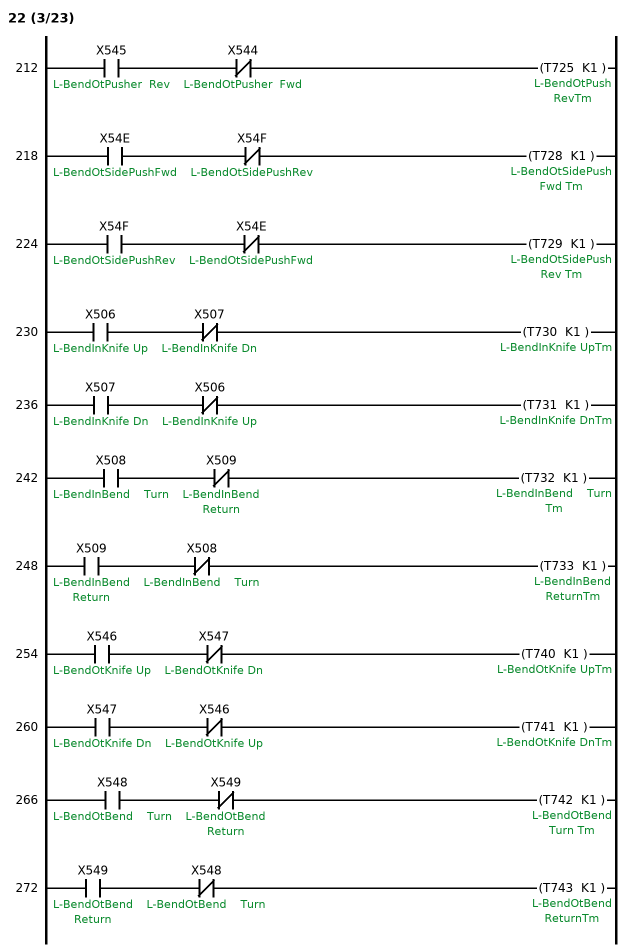
212   LD      X545  ; L-BendOtPusher  Rev
      ANI     X544  ; L-BendOtPusher  Fwd
      OUT     T725 K1  ; L-BendOtPush RevTm
218   LD      X54E  ; L-BendOtSidePushFwd
      ANI     X54F  ; L-BendOtSidePushRev
      OUT     T728 K1  ; L-BendOtSidePushFwd Tm
224   LD      X54F  ; L-BendOtSidePushRev
      ANI     X54E  ; L-BendOtSidePushFwd
      OUT     T729 K1  ; L-BendOtSidePushRev Tm
230   LD      X506  ; L-BendInKnife Up
      ANI     X507  ; L-BendInKnife Dn
      OUT     T730 K1  ; L-BendInKnife UpTm
236   LD      X507  ; L-BendInKnife Dn
      ANI     X506  ; L-BendInKnife Up
      OUT     T731 K1  ; L-BendInKnife DnTm
242   LD      X508  ; L-BendInBend    Turn
      ANI     X509  ; L-BendInBend    Return
      OUT     T732 K1  ; L-BendInBend    Turn Tm
248   LD      X509  ; L-BendInBend    Return
      ANI     X508  ; L-BendInBend    Turn
      OUT     T733 K1  ; L-BendInBend    ReturnTm
254   LD      X546  ; L-BendOtKnife Up
      ANI     X547  ; L-BendOtKnife Dn
      OUT     T740 K1  ; L-BendOtKnife UpTm
260   LD      X547  ; L-BendOtKnife Dn
      ANI     X546  ; L-BendOtKnife Up
      OUT     T741 K1  ; L-BendOtKnife DnTm
266   LD      X548  ; L-BendOtBend    Turn
      ANI     X549  ; L-BendOtBend    Return
      OUT     T742 K1  ; L-BendOtBend    Turn Tm
272   LD      X549  ; L-BendOtBend    Return
      ANI     X548  ; L-BendOtBend    Turn
      OUT     T743 K1  ; L-BendOtBend    ReturnTm
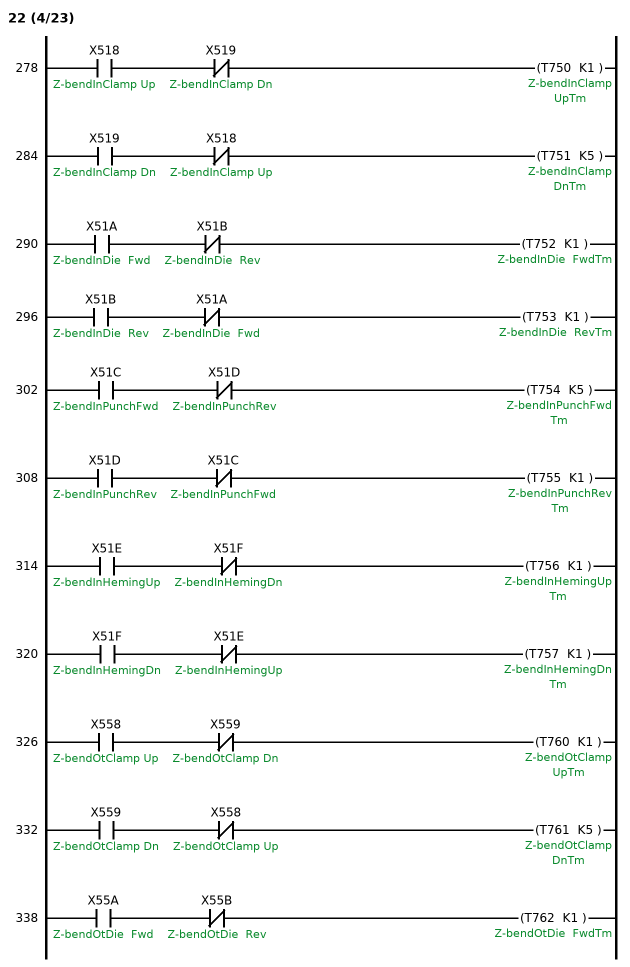
278   LD      X518  ; Z-bendInClamp Up
      ANI     X519  ; Z-bendInClamp Dn
      OUT     T750 K1  ; Z-bendInClamp UpTm
284   LD      X519  ; Z-bendInClamp Dn
      ANI     X518  ; Z-bendInClamp Up
      OUT     T751 K5  ; Z-bendInClamp DnTm
290   LD      X51A  ; Z-bendInDie  Fwd
      ANI     X51B  ; Z-bendInDie  Rev
      OUT     T752 K1  ; Z-bendInDie  FwdTm
296   LD      X51B  ; Z-bendInDie  Rev
      ANI     X51A  ; Z-bendInDie  Fwd
      OUT     T753 K1  ; Z-bendInDie  RevTm
302   LD      X51C  ; Z-bendInPunchFwd
      ANI     X51D  ; Z-bendInPunchRev
      OUT     T754 K5  ; Z-bendInPunchFwdTm
308   LD      X51D  ; Z-bendInPunchRev
      ANI     X51C  ; Z-bendInPunchFwd
      OUT     T755 K1  ; Z-bendInPunchRevTm
314   LD      X51E  ; Z-bendInHemingUp
      ANI     X51F  ; Z-bendInHemingDn
      OUT     T756 K1  ; Z-bendInHemingUpTm
320   LD      X51F  ; Z-bendInHemingDn
      ANI     X51E  ; Z-bendInHemingUp
      OUT     T757 K1  ; Z-bendInHemingDnTm
326   LD      X558  ; Z-bendOtClamp Up
      ANI     X559  ; Z-bendOtClamp Dn
      OUT     T760 K1  ; Z-bendOtClamp UpTm
332   LD      X559  ; Z-bendOtClamp Dn
      ANI     X558  ; Z-bendOtClamp Up
      OUT     T761 K5  ; Z-bendOtClamp DnTm
338   LD      X55A  ; Z-bendOtDie  Fwd
      ANI     X55B  ; Z-bendOtDie  Rev
      OUT     T762 K1  ; Z-bendOtDie  FwdTm
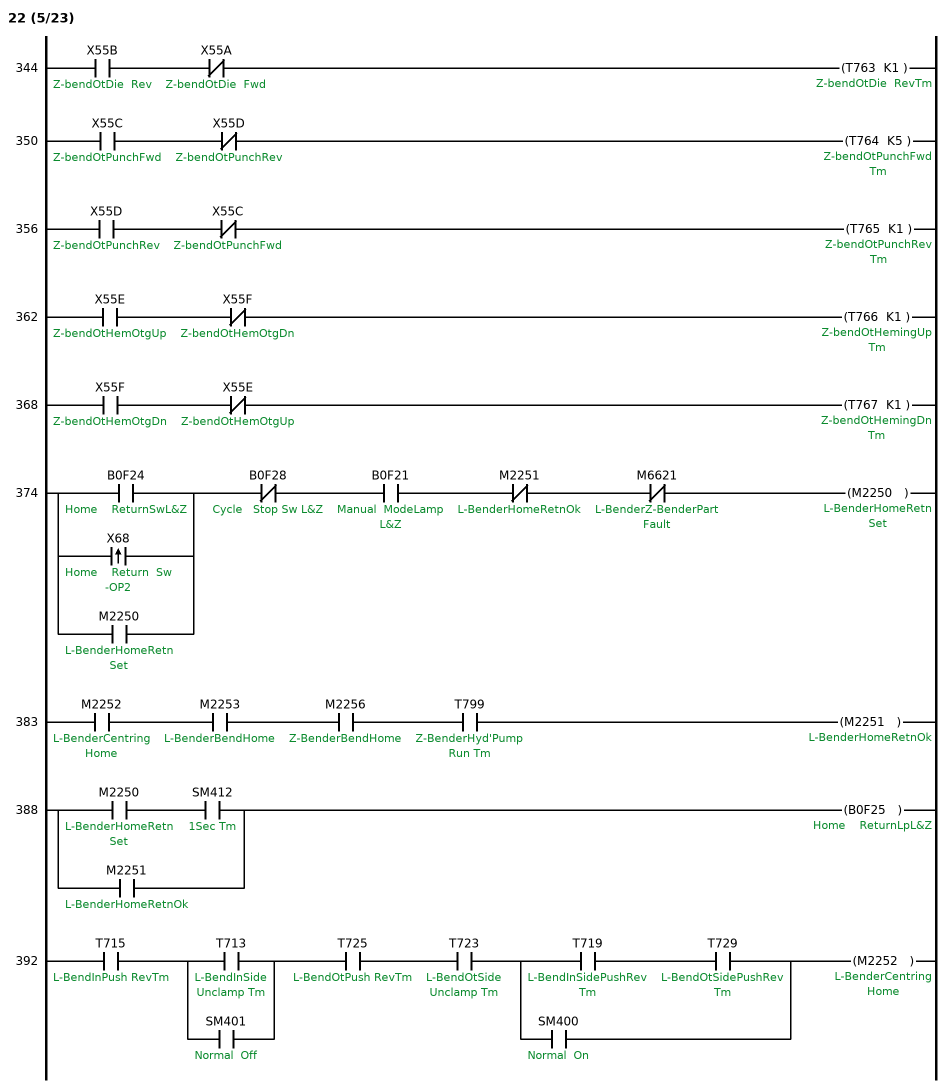
344   LD      X55B  ; Z-bendOtDie  Rev
      ANI     X55A  ; Z-bendOtDie  Fwd
      OUT     T763 K1  ; Z-bendOtDie  RevTm
350   LD      X55C  ; Z-bendOtPunchFwd
      ANI     X55D  ; Z-bendOtPunchRev
      OUT     T764 K5  ; Z-bendOtPunchFwdTm
356   LD      X55D  ; Z-bendOtPunchRev
      ANI     X55C  ; Z-bendOtPunchFwd
      OUT     T765 K1  ; Z-bendOtPunchRevTm
362   LD      X55E  ; Z-bendOtHemOtgUp
      ANI     X55F  ; Z-bendOtHemOtgDn
      OUT     T766 K1  ; Z-bendOtHemingUpTm
368   LD      X55F  ; Z-bendOtHemOtgDn
      ANI     X55E  ; Z-bendOtHemOtgUp
      OUT     T767 K1  ; Z-bendOtHemingDnTm
374   LD      B0F24  ; Home    ReturnSwL&Z
      ORP     X68  ; Home    Return  Sw -OP2
      OR      M2250  ; L-BenderHomeRetnSet
      ANI     B0F28  ; Cycle   Stop Sw L&Z
      AND     B0F21  ; Manual  ModeLampL&Z
      ANI     M2251  ; L-BenderHomeRetnOk
      ANI     M6621  ; L-BenderZ-BenderPart    Fault
      OUT     M2250  ; L-BenderHomeRetnSet
383   LD      M2252  ; L-BenderCentringHome
      AND     M2253  ; L-BenderBendHome
      AND     M2256  ; Z-BenderBendHome
      AND     T799  ; Z-BenderHyd'PumpRun Tm
      OUT     M2251  ; L-BenderHomeRetnOk
388   LD      M2250  ; L-BenderHomeRetnSet
      AND     SM412  ; 1Sec Tm
      OR      M2251  ; L-BenderHomeRetnOk
      OUT     B0F25  ; Home    ReturnLpL&Z
392   LD      T715  ; L-BendInPush RevTm
      LD      T713  ; L-BendInSide    Unclamp Tm
      OR      SM401  ; Normal  Off
      ANB
      AND     T725  ; L-BendOtPush RevTm
      AND     T723  ; L-BendOtSide    Unclamp Tm
      LD      T719  ; L-BendInSidePushRev Tm
      AND     T729  ; L-BendOtSidePushRev Tm
      OR      SM400  ; Normal  On
      ANB
      OUT     M2252  ; L-BenderCentringHome
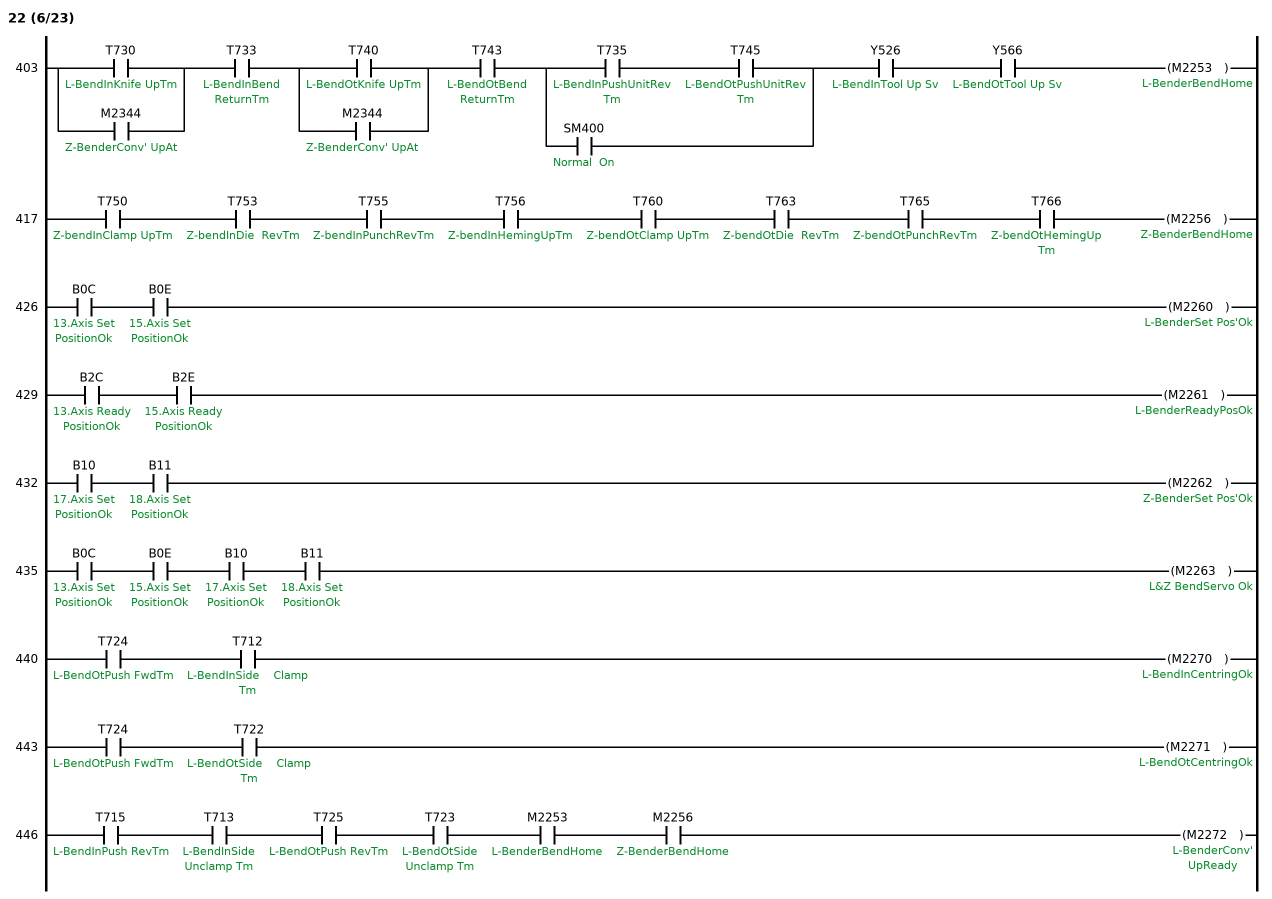
403   LD      T730  ; L-BendInKnife UpTm
      OR      M2344  ; Z-BenderConv' UpAt
      AND     T733  ; L-BendInBend    ReturnTm
      LD      T740  ; L-BendOtKnife UpTm
      OR      M2344  ; Z-BenderConv' UpAt
      ANB
      AND     T743  ; L-BendOtBend    ReturnTm
      LD      T735  ; L-BendInPushUnitRev Tm
      AND     T745  ; L-BendOtPushUnitRev Tm
      OR      SM400  ; Normal  On
      ANB
      AND     Y526  ; L-BendInTool Up Sv
      AND     Y566  ; L-BendOtTool Up Sv
      OUT     M2253  ; L-BenderBendHome
417   LD      T750  ; Z-bendInClamp UpTm
      AND     T753  ; Z-bendInDie  RevTm
      AND     T755  ; Z-bendInPunchRevTm
      AND     T756  ; Z-bendInHemingUpTm
      AND     T760  ; Z-bendOtClamp UpTm
      AND     T763  ; Z-bendOtDie  RevTm
      AND     T765  ; Z-bendOtPunchRevTm
      AND     T766  ; Z-bendOtHemingUpTm
      OUT     M2256  ; Z-BenderBendHome
426   LD      B0C  ; 13.Axis Set     PositionOk
      AND     B0E  ; 15.Axis Set     PositionOk
      OUT     M2260  ; L-BenderSet Pos'Ok
429   LD      B2C  ; 13.Axis Ready   PositionOk
      AND     B2E  ; 15.Axis Ready   PositionOk
      OUT     M2261  ; L-BenderReadyPosOk
432   LD      B10  ; 17.Axis Set     PositionOk
      AND     B11  ; 18.Axis Set     PositionOk
      OUT     M2262  ; Z-BenderSet Pos'Ok
435   LD      B0C  ; 13.Axis Set     PositionOk
      AND     B0E  ; 15.Axis Set     PositionOk
      AND     B10  ; 17.Axis Set     PositionOk
      AND     B11  ; 18.Axis Set     PositionOk
      OUT     M2263  ; L&Z BendServo Ok
440   LD      T724  ; L-BendOtPush FwdTm
      AND     T712  ; L-BendInSide    Clamp Tm
      OUT     M2270  ; L-BendInCentringOk
443   LD      T724  ; L-BendOtPush FwdTm
      AND     T722  ; L-BendOtSide    Clamp Tm
      OUT     M2271  ; L-BendOtCentringOk
446   LD      T715  ; L-BendInPush RevTm
      AND     T713  ; L-BendInSide    Unclamp Tm
      AND     T725  ; L-BendOtPush RevTm
      AND     T723  ; L-BendOtSide    Unclamp Tm
      AND     M2253  ; L-BenderBendHome
      AND     M2256  ; Z-BenderBendHome
      OUT     M2272  ; L-BenderConv' UpReady
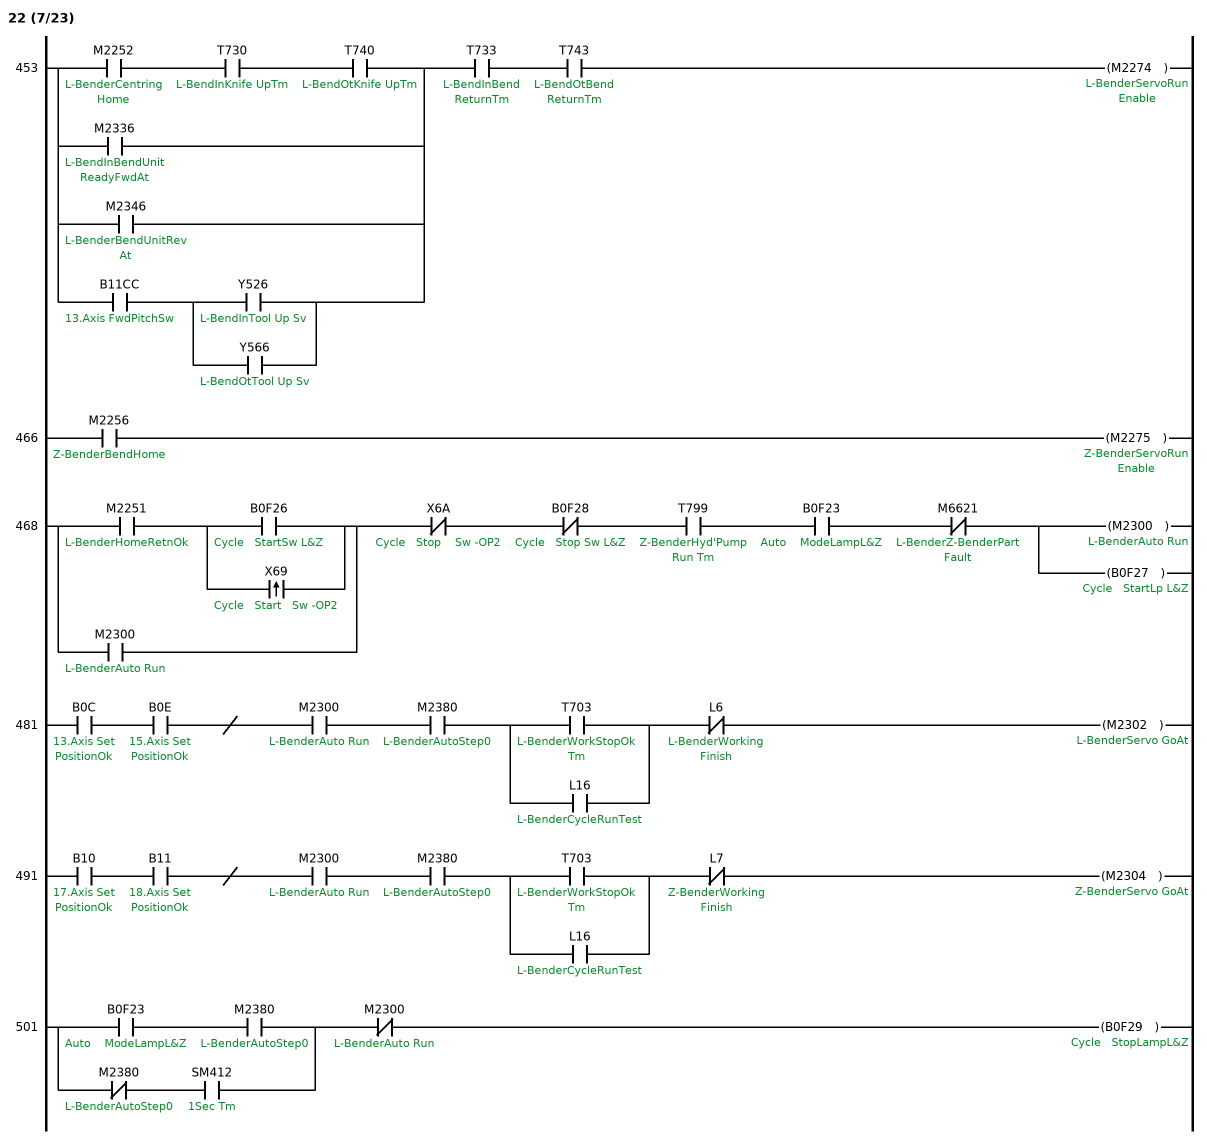
453   LD      M2252  ; L-BenderCentringHome
      AND     T730  ; L-BendInKnife UpTm
      AND     T740  ; L-BendOtKnife UpTm
      OR      M2336  ; L-BendInBendUnitReadyFwdAt
      OR      M2346  ; L-BenderBendUnitRev At
      LD      B11CC  ; 13.Axis FwdPitchSw
      LD      Y526  ; L-BendInTool Up Sv
      OR      Y566  ; L-BendOtTool Up Sv
      ANB
      ORB
      AND     T733  ; L-BendInBend    ReturnTm
      AND     T743  ; L-BendOtBend    ReturnTm
      OUT     M2274  ; L-BenderServoRunEnable
466   LD      M2256  ; Z-BenderBendHome
      OUT     M2275  ; Z-BenderServoRunEnable
468   LD      M2251  ; L-BenderHomeRetnOk
      LD      B0F26  ; Cycle   StartSw L&Z
      ORP     X69  ; Cycle   Start   Sw -OP2
      ANB
      OR      M2300  ; L-BenderAuto Run
      ANI     X6A  ; Cycle   Stop    Sw -OP2
      ANI     B0F28  ; Cycle   Stop Sw L&Z
      AND     T799  ; Z-BenderHyd'PumpRun Tm
      AND     B0F23  ; Auto    ModeLampL&Z
      ANI     M6621  ; L-BenderZ-BenderPart    Fault
      OUT     M2300  ; L-BenderAuto Run
      OUT     B0F27  ; Cycle   StartLp L&Z
481   LD      B0C  ; 13.Axis Set     PositionOk
      AND     B0E  ; 15.Axis Set     PositionOk
      INV
      AND     M2300  ; L-BenderAuto Run
      AND     M2380  ; L-BenderAutoStep0
      LD      T703  ; L-BenderWorkStopOk Tm
      OR      L16  ; L-BenderCycleRunTest
      ANB
      ANI     L6  ; L-BenderWorking Finish
      OUT     M2302  ; L-BenderServo GoAt
491   LD      B10  ; 17.Axis Set     PositionOk
      AND     B11  ; 18.Axis Set     PositionOk
      INV
      AND     M2300  ; L-BenderAuto Run
      AND     M2380  ; L-BenderAutoStep0
      LD      T703  ; L-BenderWorkStopOk Tm
      OR      L16  ; L-BenderCycleRunTest
      ANB
      ANI     L7  ; Z-BenderWorking Finish
      OUT     M2304  ; Z-BenderServo GoAt
501   LD      B0F23  ; Auto    ModeLampL&Z
      AND     M2380  ; L-BenderAutoStep0
      LDI     M2380  ; L-BenderAutoStep0
      AND     SM412  ; 1Sec Tm
      ORB
      ANI     M2300  ; L-BenderAuto Run
      OUT     B0F29  ; Cycle   StopLampL&Z
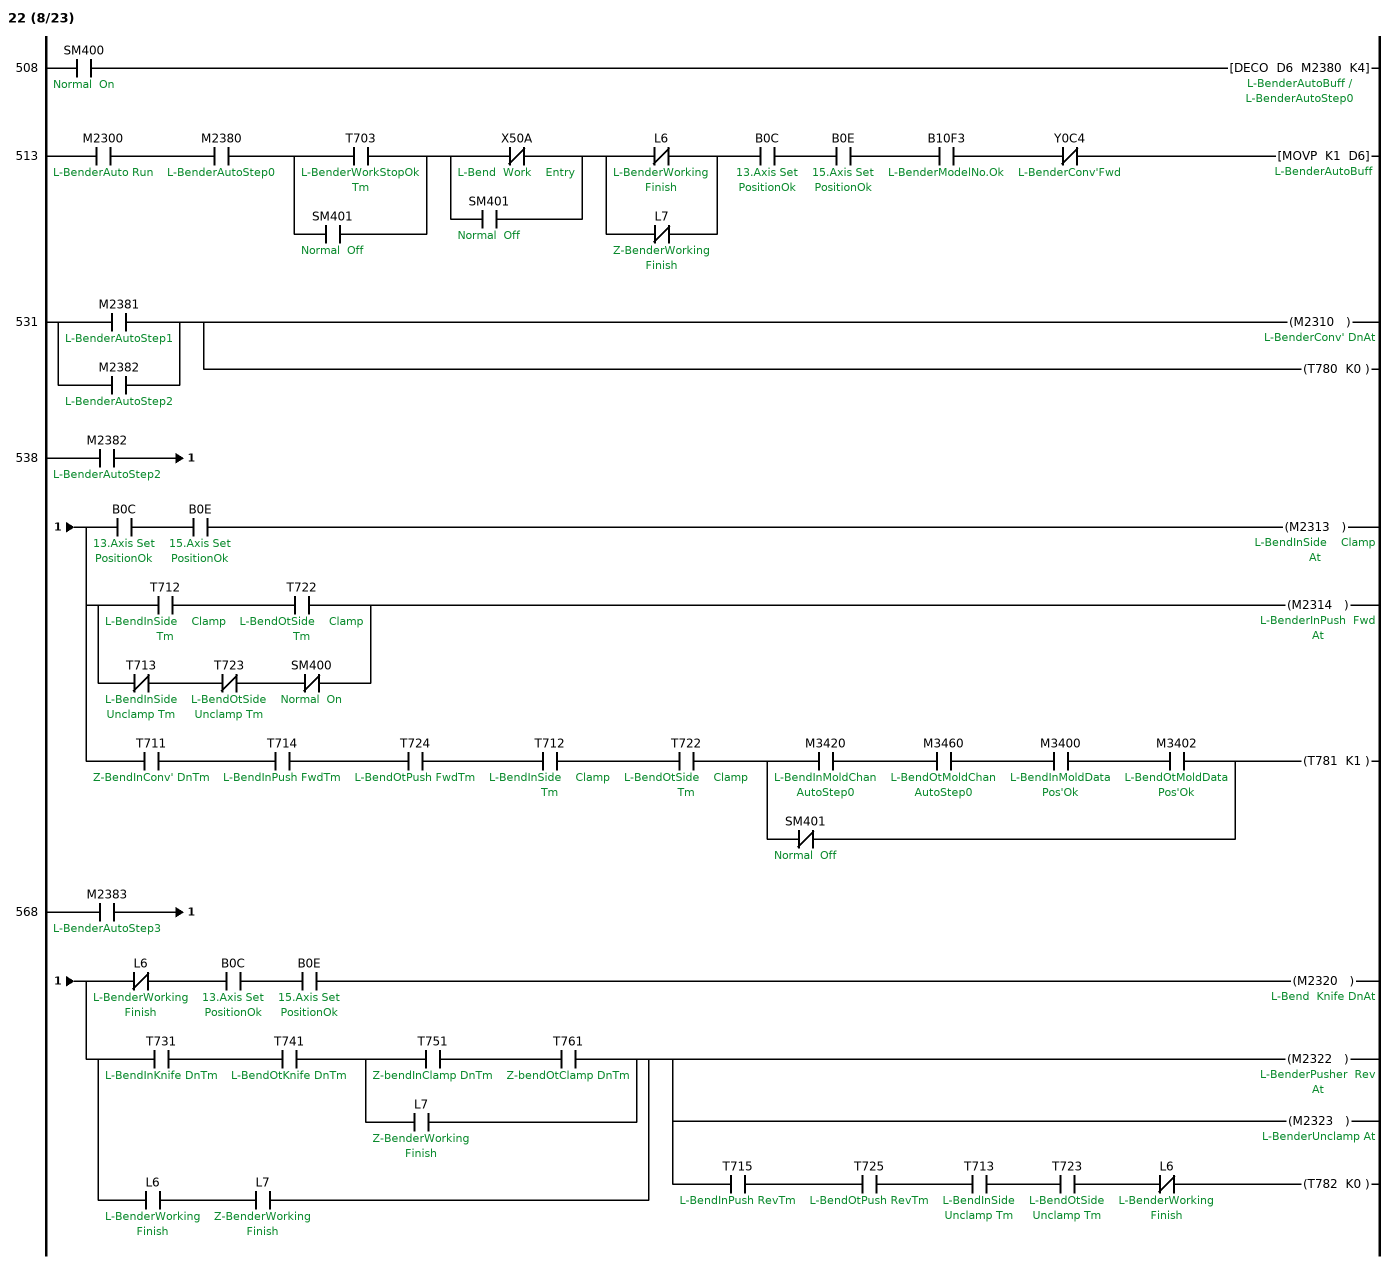
508   LD      SM400  ; Normal  On
      DECO    D6 M2380 K4  ; L-BenderAutoBuff
513   LD      M2300  ; L-BenderAuto Run
      AND     M2380  ; L-BenderAutoStep0
      LD      T703  ; L-BenderWorkStopOk Tm
      OR      SM401  ; Normal  Off
      ANB
      LDI     X50A  ; L-Bend  Work    Entry
      OR      SM401  ; Normal  Off
      ANB
      LDI     L6  ; L-BenderWorking Finish
      ORI     L7  ; Z-BenderWorking Finish
      ANB
      AND     B0C  ; 13.Axis Set     PositionOk
      AND     B0E  ; 15.Axis Set     PositionOk
      AND     B10F3  ; L-BenderModelNo.Ok
      ANI     Y0C4  ; L-BenderConv'Fwd
      MOVP    K1 D6
531   LD      M2381  ; L-BenderAutoStep1
      OR      M2382  ; L-BenderAutoStep2
      OUT     M2310  ; L-BenderConv' DnAt
      OUT     T780 K0
538   LD      M2382  ; L-BenderAutoStep2
      MPS
      AND     B0C  ; 13.Axis Set     PositionOk
      AND     B0E  ; 15.Axis Set     PositionOk
      OUT     M2313  ; L-BendInSide    Clamp At
      MRD
      LD      T712  ; L-BendInSide    Clamp Tm
      AND     T722  ; L-BendOtSide    Clamp Tm
      LDI     T713  ; L-BendInSide    Unclamp Tm
      ANI     T723  ; L-BendOtSide    Unclamp Tm
      ANI     SM400  ; Normal  On
      ORB
      ANB
      OUT     M2314  ; L-BenderInPush  Fwd At
      MPP
      AND     T711  ; Z-BendInConv' DnTm
      AND     T714  ; L-BendInPush FwdTm
      AND     T724  ; L-BendOtPush FwdTm
      AND     T712  ; L-BendInSide    Clamp Tm
      AND     T722  ; L-BendOtSide    Clamp Tm
      LD      M3420  ; L-BendInMoldChanAutoStep0
      AND     M3460  ; L-BendOtMoldChanAutoStep0
      AND     M3400  ; L-BendInMoldDataPos'Ok
      AND     M3402  ; L-BendOtMoldDataPos'Ok
      ORI     SM401  ; Normal  Off
      ANB
      OUT     T781 K1
568   LD      M2383  ; L-BenderAutoStep3
      MPS
      ANI     L6  ; L-BenderWorking Finish
      AND     B0C  ; 13.Axis Set     PositionOk
      AND     B0E  ; 15.Axis Set     PositionOk
      OUT     M2320  ; L-Bend  Knife DnAt
      MPP
      LD      T731  ; L-BendInKnife DnTm
      AND     T741  ; L-BendOtKnife DnTm
      LD      T751  ; Z-bendInClamp DnTm
      AND     T761  ; Z-bendOtClamp DnTm
      OR      L7  ; Z-BenderWorking Finish
      ANB
      LD      L6  ; L-BenderWorking Finish
      AND     L7  ; Z-BenderWorking Finish
      ORB
      ANB
      OUT     M2322  ; L-BenderPusher  Rev At
      OUT     M2323  ; L-BenderUnclamp At
      AND     T715  ; L-BendInPush RevTm
      AND     T725  ; L-BendOtPush RevTm
      AND     T713  ; L-BendInSide    Unclamp Tm
      AND     T723  ; L-BendOtSide    Unclamp Tm
      ANI     L6  ; L-BenderWorking Finish
      OUT     T782 K0
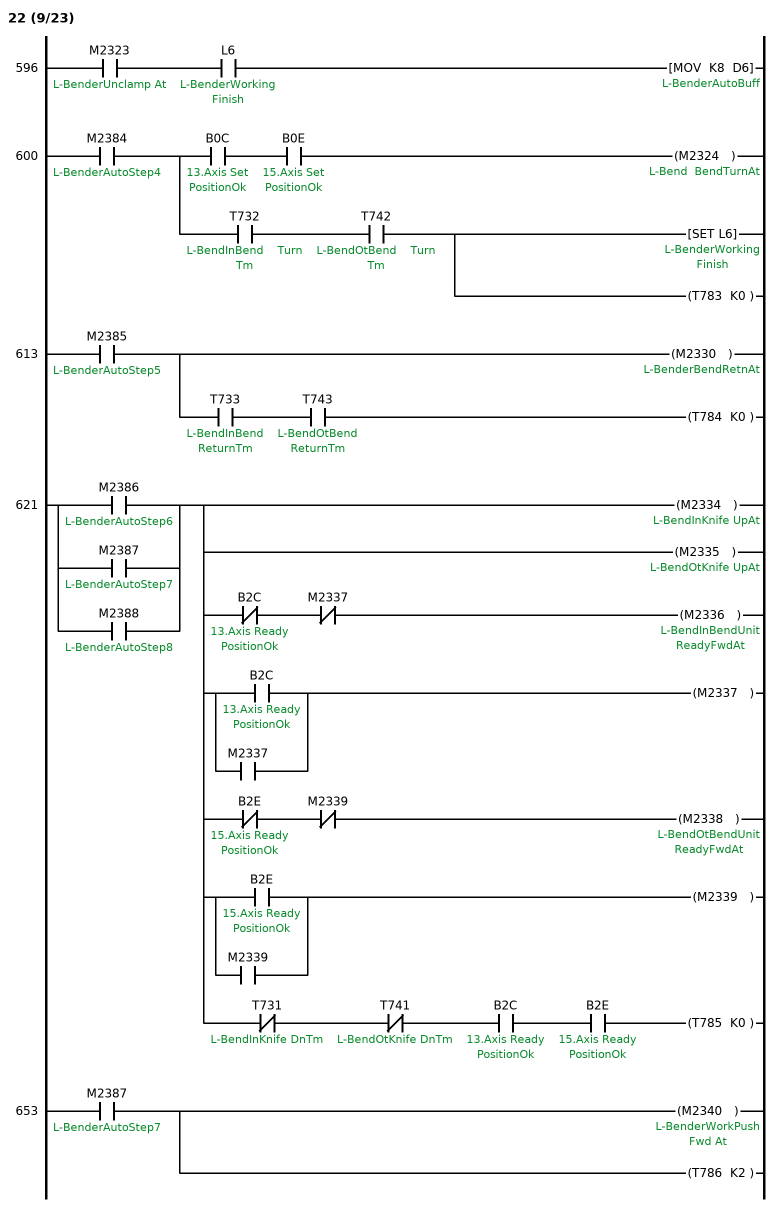
596   LD      M2323  ; L-BenderUnclamp At
      AND     L6  ; L-BenderWorking Finish
      MOV     K8 D6
600   LD      M2384  ; L-BenderAutoStep4
      MPS
      AND     B0C  ; 13.Axis Set     PositionOk
      AND     B0E  ; 15.Axis Set     PositionOk
      OUT     M2324  ; L-Bend  BendTurnAt
      MPP
      AND     T732  ; L-BendInBend    Turn Tm
      AND     T742  ; L-BendOtBend    Turn Tm
      SET     L6  ; L-BenderWorking Finish
      OUT     T783 K0
613   LD      M2385  ; L-BenderAutoStep5
      OUT     M2330  ; L-BenderBendRetnAt
      AND     T733  ; L-BendInBend    ReturnTm
      AND     T743  ; L-BendOtBend    ReturnTm
      OUT     T784 K0
621   LD      M2386  ; L-BenderAutoStep6
      OR      M2387  ; L-BenderAutoStep7
      OR      M2388  ; L-BenderAutoStep8
      OUT     M2334  ; L-BendInKnife UpAt
      OUT     M2335  ; L-BendOtKnife UpAt
      MPS
      ANI     B2C  ; 13.Axis Ready   PositionOk
      ANI     M2337
      OUT     M2336  ; L-BendInBendUnitReadyFwdAt
      MRD
      LD      B2C  ; 13.Axis Ready   PositionOk
      OR      M2337
      ANB
      OUT     M2337
      MRD
      ANI     B2E  ; 15.Axis Ready   PositionOk
      ANI     M2339
      OUT     M2338  ; L-BendOtBendUnitReadyFwdAt
      MRD
      LD      B2E  ; 15.Axis Ready   PositionOk
      OR      M2339
      ANB
      OUT     M2339
      MPP
      ANI     T731  ; L-BendInKnife DnTm
      ANI     T741  ; L-BendOtKnife DnTm
      AND     B2C  ; 13.Axis Ready   PositionOk
      AND     B2E  ; 15.Axis Ready   PositionOk
      OUT     T785 K0
653   LD      M2387  ; L-BenderAutoStep7
      OUT     M2340  ; L-BenderWorkPushFwd At
      OUT     T786 K2
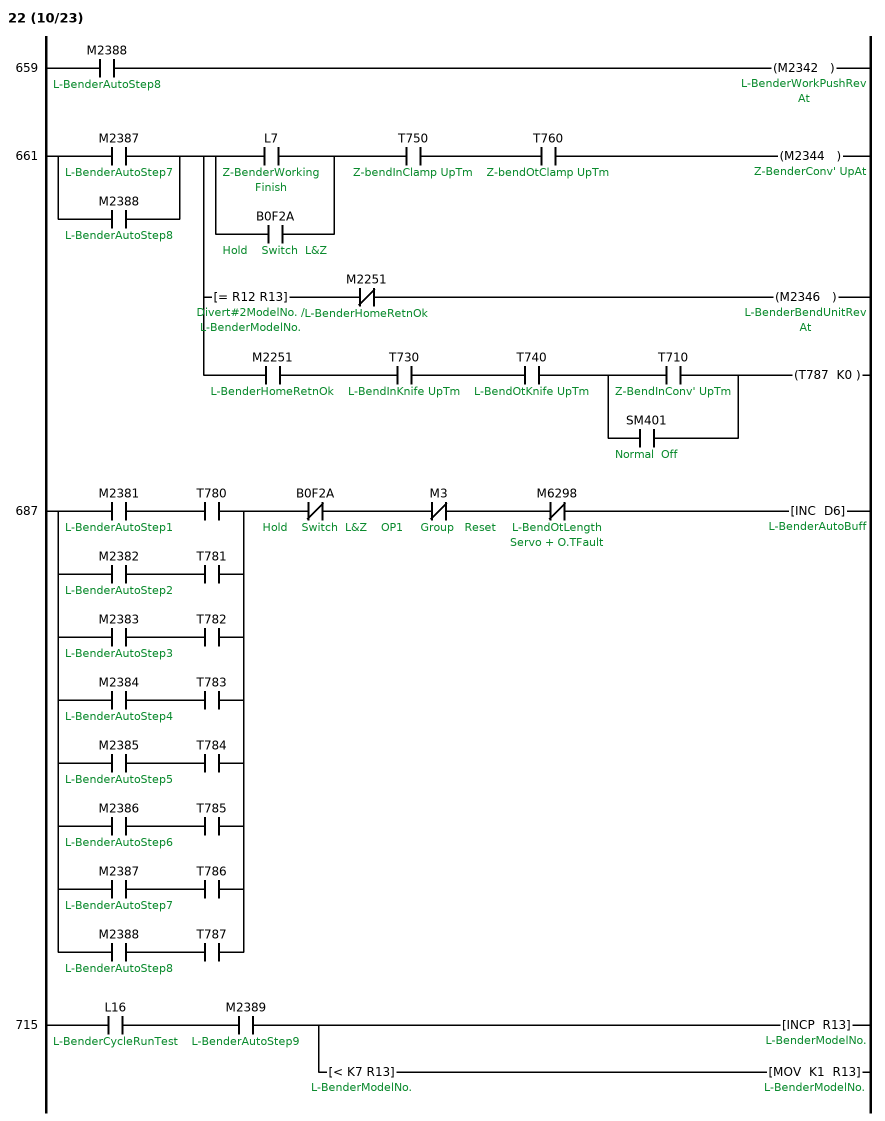
659   LD      M2388  ; L-BenderAutoStep8
      OUT     M2342  ; L-BenderWorkPushRev At
661   LD      M2387  ; L-BenderAutoStep7
      OR      M2388  ; L-BenderAutoStep8
      MPS
      LD      L7  ; Z-BenderWorking Finish
      OR      B0F2A  ; Hold    Switch  L&Z
      ANB
      AND     T750  ; Z-bendInClamp UpTm
      AND     T760  ; Z-bendOtClamp UpTm
      OUT     M2344  ; Z-BenderConv' UpAt
      MRD
      AND=    R12 R13  ; Divert#2ModelNo. / L-BenderModelNo.
      ANI     M2251  ; L-BenderHomeRetnOk
      OUT     M2346  ; L-BenderBendUnitRev At
      MPP
      AND     M2251  ; L-BenderHomeRetnOk
      AND     T730  ; L-BendInKnife UpTm
      AND     T740  ; L-BendOtKnife UpTm
      LD      T710  ; Z-BendInConv' UpTm
      OR      SM401  ; Normal  Off
      ANB
      OUT     T787 K0
687   LD      M2381  ; L-BenderAutoStep1
      AND     T780
      LD      M2382  ; L-BenderAutoStep2
      AND     T781
      ORB
      LD      M2383  ; L-BenderAutoStep3
      AND     T782
      ORB
      LD      M2384  ; L-BenderAutoStep4
      AND     T783
      ORB
      LD      M2385  ; L-BenderAutoStep5
      AND     T784
      ORB
      LD      M2386  ; L-BenderAutoStep6
      AND     T785
      ORB
      LD      M2387  ; L-BenderAutoStep7
      AND     T786
      ORB
      LD      M2388  ; L-BenderAutoStep8
      AND     T787
      ORB
      ANI     B0F2A  ; Hold    Switch  L&Z
      ANI     M3  ; OP1     Group   Reset
      ANI     M6298  ; L-BendOtLength  Servo + O.TFault
      INC     D6
715   LD      L16  ; L-BenderCycleRunTest
      AND     M2389  ; L-BenderAutoStep9
      INCP    R13
      AND<    K7 R13  ; L-BenderModelNo.
      MOV     K1 R13
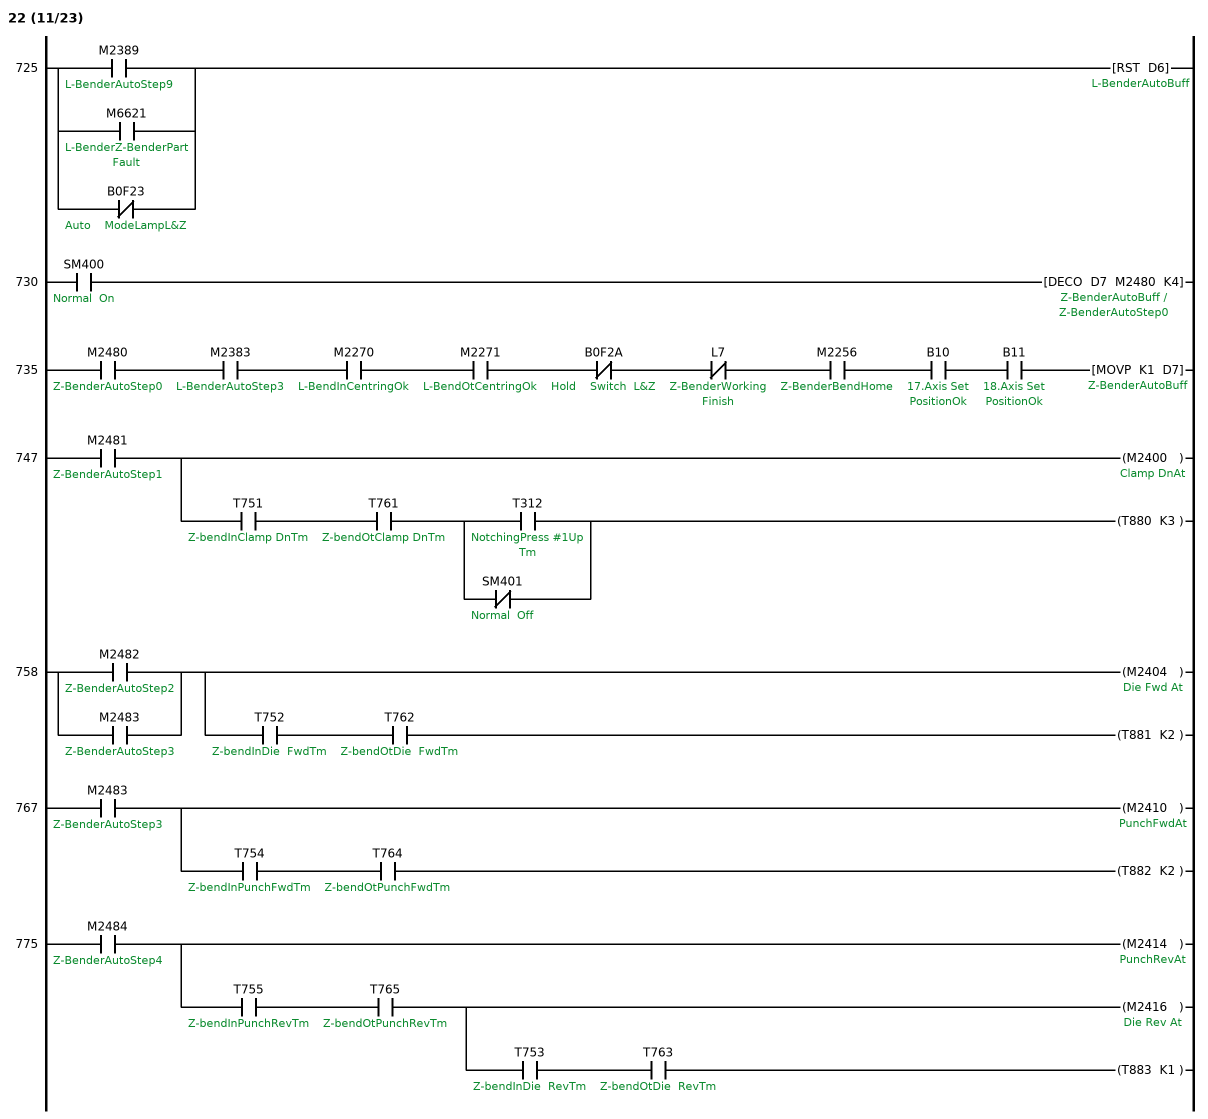
725   LD      M2389  ; L-BenderAutoStep9
      OR      M6621  ; L-BenderZ-BenderPart    Fault
      ORI     B0F23  ; Auto    ModeLampL&Z
      RST     D6  ; L-BenderAutoBuff
730   LD      SM400  ; Normal  On
      DECO    D7 M2480 K4  ; Z-BenderAutoBuff / Z-BenderAutoStep0
735   LD      M2480  ; Z-BenderAutoStep0
      AND     M2383  ; L-BenderAutoStep3
      AND     M2270  ; L-BendInCentringOk
      AND     M2271  ; L-BendOtCentringOk
      ANI     B0F2A  ; Hold    Switch  L&Z
      ANI     L7  ; Z-BenderWorking Finish
      AND     M2256  ; Z-BenderBendHome
      AND     B10  ; 17.Axis Set     PositionOk
      AND     B11  ; 18.Axis Set     PositionOk
      MOVP    K1 D7
747   LD      M2481  ; Z-BenderAutoStep1
      OUT     M2400  ; Clamp DnAt
      AND     T751  ; Z-bendInClamp DnTm
      AND     T761  ; Z-bendOtClamp DnTm
      LD      T312  ; NotchingPress #1Up Tm
      ORI     SM401  ; Normal  Off
      ANB
      OUT     T880 K3
758   LD      M2482  ; Z-BenderAutoStep2
      OR      M2483  ; Z-BenderAutoStep3
      OUT     M2404  ; Die Fwd At
      AND     T752  ; Z-bendInDie  FwdTm
      AND     T762  ; Z-bendOtDie  FwdTm
      OUT     T881 K2
767   LD      M2483  ; Z-BenderAutoStep3
      OUT     M2410  ; PunchFwdAt
      AND     T754  ; Z-bendInPunchFwdTm
      AND     T764  ; Z-bendOtPunchFwdTm
      OUT     T882 K2
775   LD      M2484  ; Z-BenderAutoStep4
      OUT     M2414  ; PunchRevAt
      AND     T755  ; Z-bendInPunchRevTm
      AND     T765  ; Z-bendOtPunchRevTm
      OUT     M2416  ; Die Rev At
      AND     T753  ; Z-bendInDie  RevTm
      AND     T763  ; Z-bendOtDie  RevTm
      OUT     T883 K1
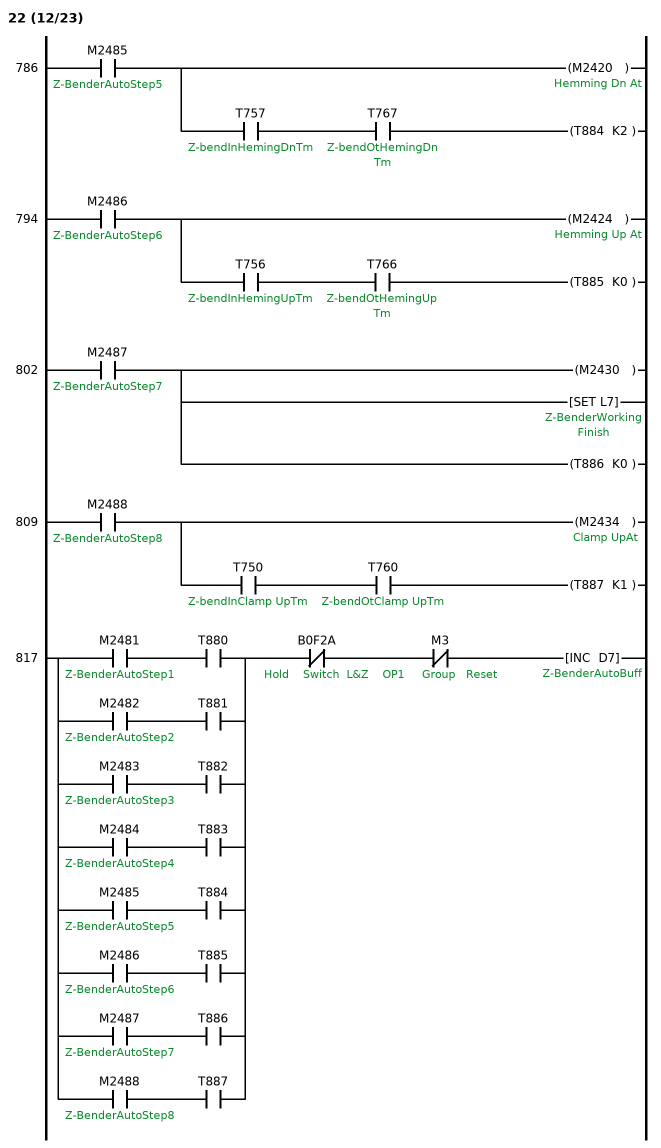
786   LD      M2485  ; Z-BenderAutoStep5
      OUT     M2420  ; Hemming Dn At
      AND     T757  ; Z-bendInHemingDnTm
      AND     T767  ; Z-bendOtHemingDnTm
      OUT     T884 K2
794   LD      M2486  ; Z-BenderAutoStep6
      OUT     M2424  ; Hemming Up At
      AND     T756  ; Z-bendInHemingUpTm
      AND     T766  ; Z-bendOtHemingUpTm
      OUT     T885 K0
802   LD      M2487  ; Z-BenderAutoStep7
      OUT     M2430
      SET     L7  ; Z-BenderWorking Finish
      OUT     T886 K0
809   LD      M2488  ; Z-BenderAutoStep8
      OUT     M2434  ; Clamp UpAt
      AND     T750  ; Z-bendInClamp UpTm
      AND     T760  ; Z-bendOtClamp UpTm
      OUT     T887 K1
817   LD      M2481  ; Z-BenderAutoStep1
      AND     T880
      LD      M2482  ; Z-BenderAutoStep2
      AND     T881
      ORB
      LD      M2483  ; Z-BenderAutoStep3
      AND     T882
      ORB
      LD      M2484  ; Z-BenderAutoStep4
      AND     T883
      ORB
      LD      M2485  ; Z-BenderAutoStep5
      AND     T884
      ORB
      LD      M2486  ; Z-BenderAutoStep6
      AND     T885
      ORB
      LD      M2487  ; Z-BenderAutoStep7
      AND     T886
      ORB
      LD      M2488  ; Z-BenderAutoStep8
      AND     T887
      ORB
      ANI     B0F2A  ; Hold    Switch  L&Z
      ANI     M3  ; OP1     Group   Reset
      INC     D7
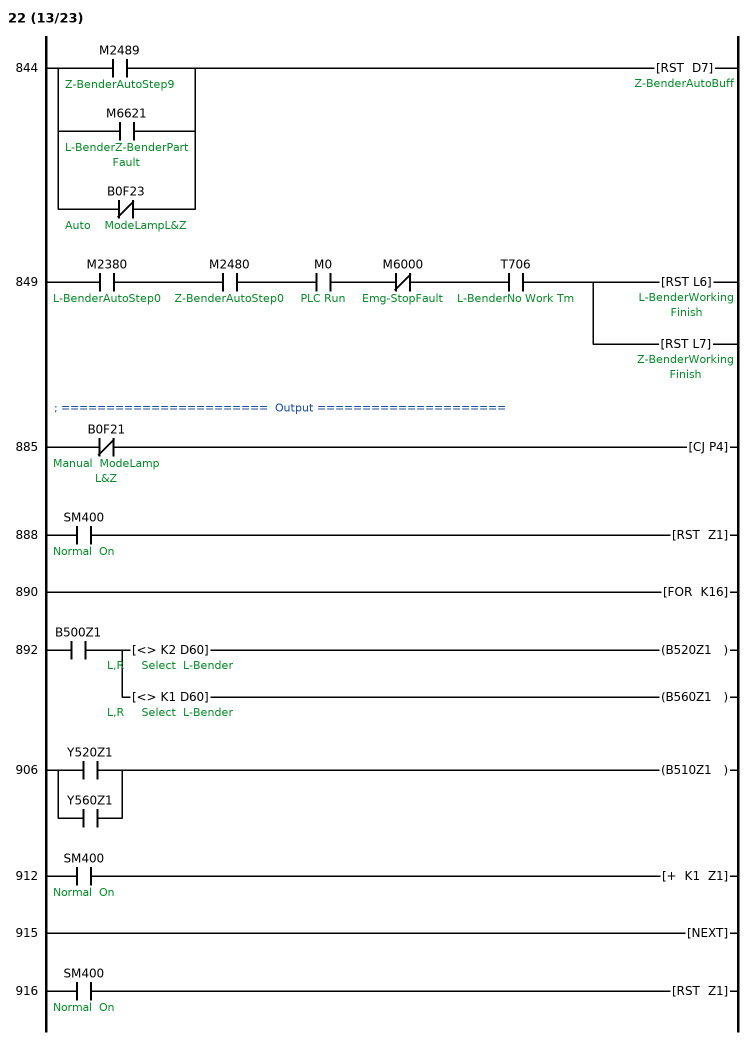
844   LD      M2489  ; Z-BenderAutoStep9
      OR      M6621  ; L-BenderZ-BenderPart    Fault
      ORI     B0F23  ; Auto    ModeLampL&Z
      RST     D7  ; Z-BenderAutoBuff
849   LD      M2380  ; L-BenderAutoStep0
      AND     M2480  ; Z-BenderAutoStep0
      AND     M0  ; PLC Run
      ANI     M6000  ; Emg-StopFault
      AND     T706  ; L-BenderNo Work Tm
      RST     L6  ; L-BenderWorking Finish
      RST     L7  ; Z-BenderWorking Finish
; =======================  Output =====================
885   LDI     B0F21  ; Manual  ModeLampL&Z
      CJ      P4
888   LD      SM400  ; Normal  On
      RST     Z1
890   FOR     K16
892   LD      B500Z1
      MPS
      AND<>   K2 D60  ; L,R     Select  L-Bender
      OUT     B520Z1
      MPP
      AND<>   K1 D60  ; L,R     Select  L-Bender
      OUT     B560Z1
906   LD      Y520Z1
      OR      Y560Z1
      OUT     B510Z1
912   LD      SM400  ; Normal  On
      +       K1 Z1
915   NEXT
916   LD      SM400  ; Normal  On
      RST     Z1
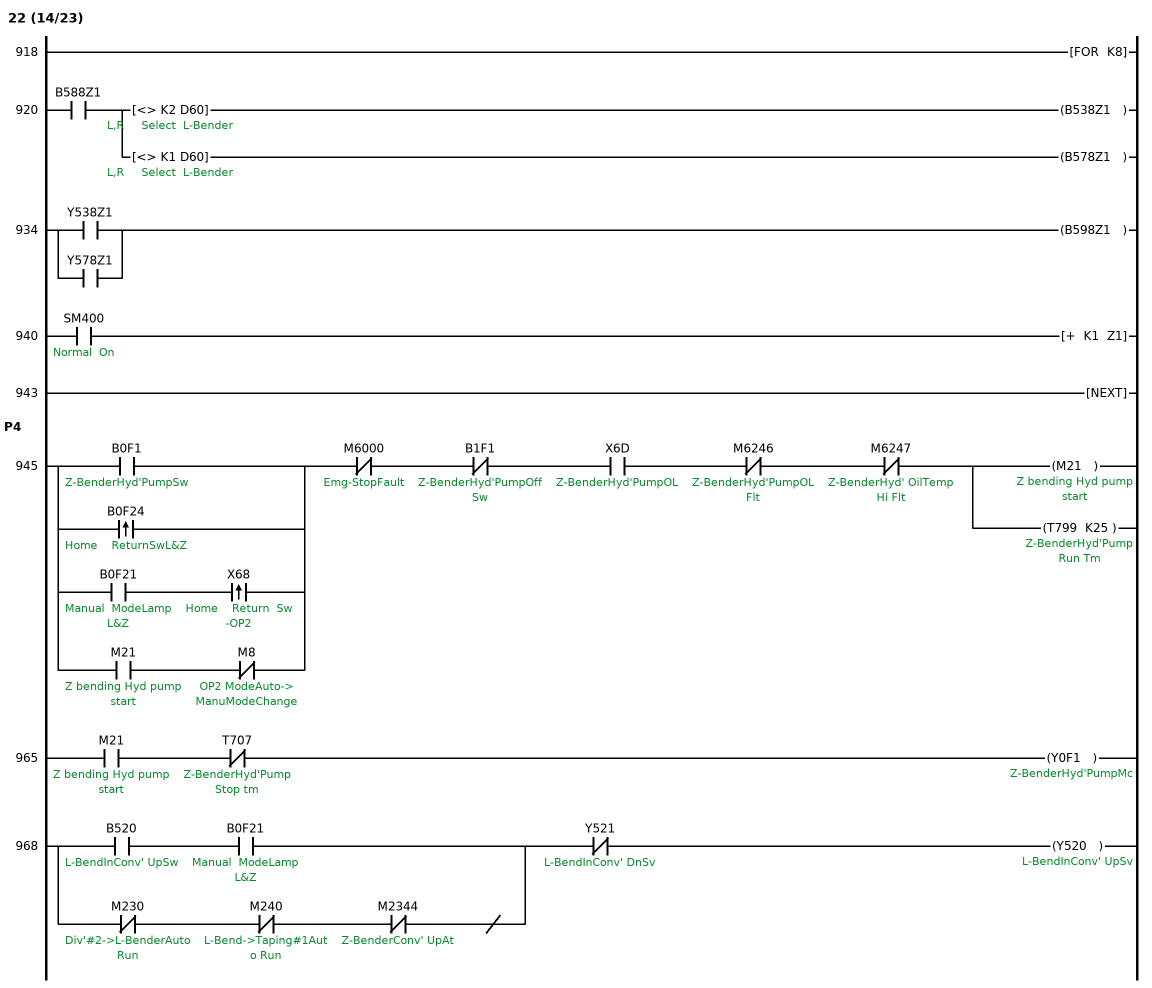
918   FOR     K8
920   LD      B588Z1
      MPS
      AND<>   K2 D60  ; L,R     Select  L-Bender
      OUT     B538Z1
      MPP
      AND<>   K1 D60  ; L,R     Select  L-Bender
      OUT     B578Z1
934   LD      Y538Z1
      OR      Y578Z1
      OUT     B598Z1
940   LD      SM400  ; Normal  On
      +       K1 Z1
943   NEXT
      P4
945   LD      B0F1  ; Z-BenderHyd'PumpSw
      ORP     B0F24  ; Home    ReturnSwL&Z
      LD      B0F21  ; Manual  ModeLampL&Z
      ANDP    X68  ; Home    Return  Sw -OP2
      ORB
      LD      M21  ; Z bending Hyd pump start
      ANI     M8  ; OP2 ModeAuto->  ManuModeChange
      ORB
      ANI     M6000  ; Emg-StopFault
      ANI     B1F1  ; Z-BenderHyd'PumpOff Sw
      AND     X6D  ; Z-BenderHyd'PumpOL
      ANI     M6246  ; Z-BenderHyd'PumpOL Flt
      ANI     M6247  ; Z-BenderHyd' OilTemp Hi Flt
      OUT     M21  ; Z bending Hyd pump start
      OUT     T799 K25  ; Z-BenderHyd'PumpRun Tm
965   LD      M21  ; Z bending Hyd pump start
      ANI     T707  ; Z-BenderHyd'PumpStop tm
      OUT     Y0F1  ; Z-BenderHyd'PumpMc
968   LD      B520  ; L-BendInConv' UpSw
      AND     B0F21  ; Manual  ModeLampL&Z
      LDI     M230  ; Div'#2->L-BenderAuto Run
      ANI     M240  ; L-Bend->Taping#1Auto Run
      ANI     M2344  ; Z-BenderConv' UpAt
      INV
      ORB
      ANI     Y521  ; L-BendInConv' DnSv
      OUT     Y520  ; L-BendInConv' UpSv
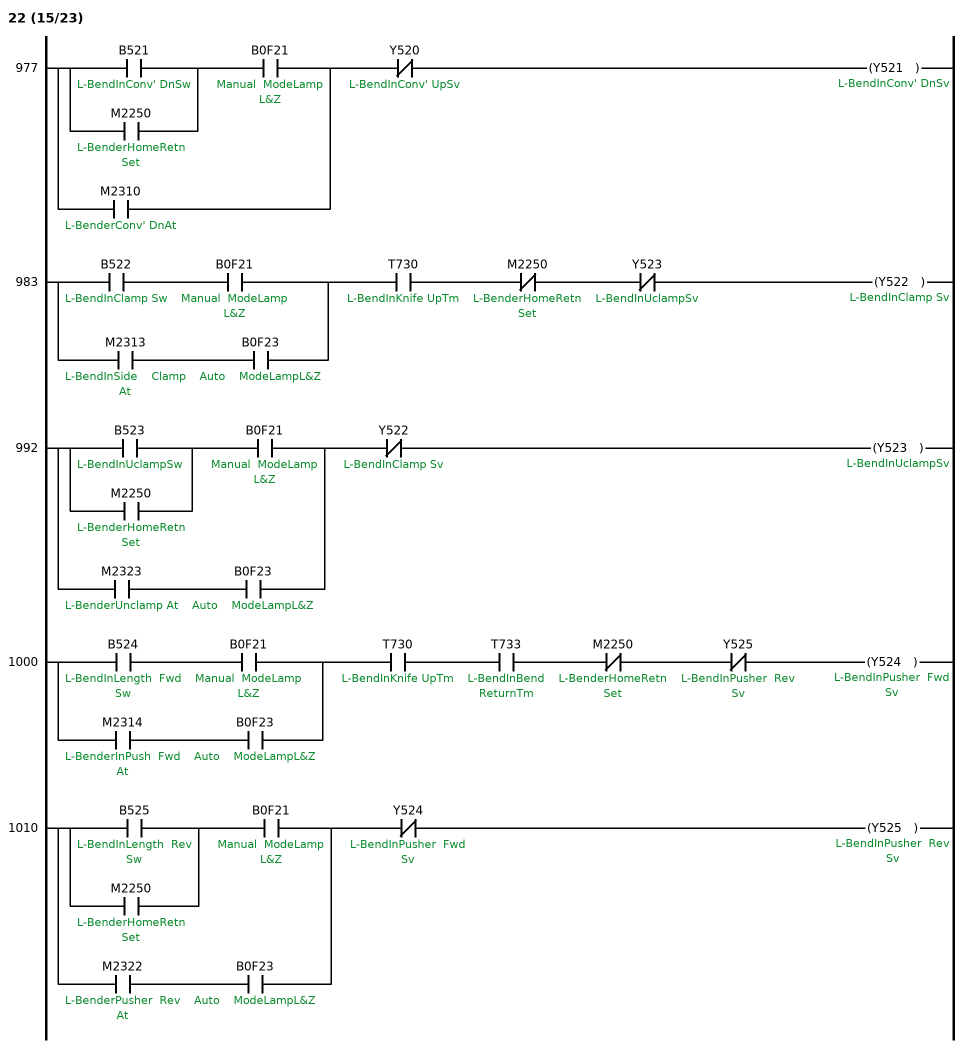
977   LD      B521  ; L-BendInConv' DnSw
      OR      M2250  ; L-BenderHomeRetnSet
      AND     B0F21  ; Manual  ModeLampL&Z
      OR      M2310  ; L-BenderConv' DnAt
      ANI     Y520  ; L-BendInConv' UpSv
      OUT     Y521  ; L-BendInConv' DnSv
983   LD      B522  ; L-BendInClamp Sw
      AND     B0F21  ; Manual  ModeLampL&Z
      LD      M2313  ; L-BendInSide    Clamp At
      AND     B0F23  ; Auto    ModeLampL&Z
      ORB
      AND     T730  ; L-BendInKnife UpTm
      ANI     M2250  ; L-BenderHomeRetnSet
      ANI     Y523  ; L-BendInUclampSv
      OUT     Y522  ; L-BendInClamp Sv
992   LD      B523  ; L-BendInUclampSw
      OR      M2250  ; L-BenderHomeRetnSet
      AND     B0F21  ; Manual  ModeLampL&Z
      LD      M2323  ; L-BenderUnclamp At
      AND     B0F23  ; Auto    ModeLampL&Z
      ORB
      ANI     Y522  ; L-BendInClamp Sv
      OUT     Y523  ; L-BendInUclampSv
1000  LD      B524  ; L-BendInLength  Fwd Sw
      AND     B0F21  ; Manual  ModeLampL&Z
      LD      M2314  ; L-BenderInPush  Fwd At
      AND     B0F23  ; Auto    ModeLampL&Z
      ORB
      AND     T730  ; L-BendInKnife UpTm
      AND     T733  ; L-BendInBend    ReturnTm
      ANI     M2250  ; L-BenderHomeRetnSet
      ANI     Y525  ; L-BendInPusher  Rev Sv
      OUT     Y524  ; L-BendInPusher  Fwd Sv
1010  LD      B525  ; L-BendInLength  Rev Sw
      OR      M2250  ; L-BenderHomeRetnSet
      AND     B0F21  ; Manual  ModeLampL&Z
      LD      M2322  ; L-BenderPusher  Rev At
      AND     B0F23  ; Auto    ModeLampL&Z
      ORB
      ANI     Y524  ; L-BendInPusher  Fwd Sv
      OUT     Y525  ; L-BendInPusher  Rev Sv
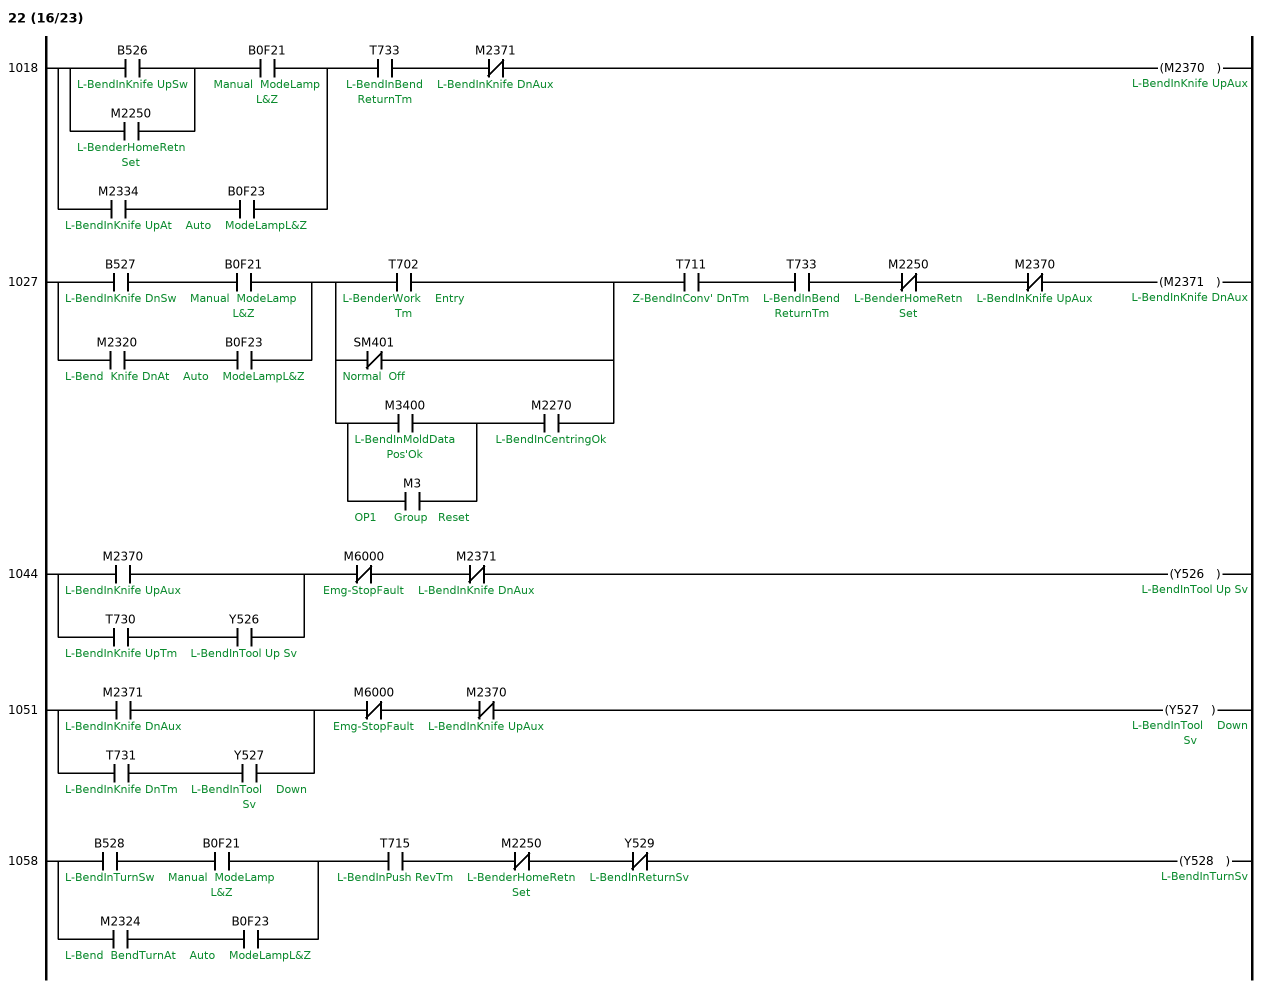
1018  LD      B526  ; L-BendInKnife UpSw
      OR      M2250  ; L-BenderHomeRetnSet
      AND     B0F21  ; Manual  ModeLampL&Z
      LD      M2334  ; L-BendInKnife UpAt
      AND     B0F23  ; Auto    ModeLampL&Z
      ORB
      AND     T733  ; L-BendInBend    ReturnTm
      ANI     M2371  ; L-BendInKnife DnAux
      OUT     M2370  ; L-BendInKnife UpAux
1027  LD      B527  ; L-BendInKnife DnSw
      AND     B0F21  ; Manual  ModeLampL&Z
      LD      M2320  ; L-Bend  Knife DnAt
      AND     B0F23  ; Auto    ModeLampL&Z
      ORB
      LD      T702  ; L-BenderWork    Entry Tm
      ORI     SM401  ; Normal  Off
      LD      M3400  ; L-BendInMoldDataPos'Ok
      OR      M3  ; OP1     Group   Reset
      AND     M2270  ; L-BendInCentringOk
      ORB
      ANB
      AND     T711  ; Z-BendInConv' DnTm
      AND     T733  ; L-BendInBend    ReturnTm
      ANI     M2250  ; L-BenderHomeRetnSet
      ANI     M2370  ; L-BendInKnife UpAux
      OUT     M2371  ; L-BendInKnife DnAux
1044  LD      M2370  ; L-BendInKnife UpAux
      LD      T730  ; L-BendInKnife UpTm
      AND     Y526  ; L-BendInTool Up Sv
      ORB
      ANI     M6000  ; Emg-StopFault
      ANI     M2371  ; L-BendInKnife DnAux
      OUT     Y526  ; L-BendInTool Up Sv
1051  LD      M2371  ; L-BendInKnife DnAux
      LD      T731  ; L-BendInKnife DnTm
      AND     Y527  ; L-BendInTool    Down Sv
      ORB
      ANI     M6000  ; Emg-StopFault
      ANI     M2370  ; L-BendInKnife UpAux
      OUT     Y527  ; L-BendInTool    Down Sv
1058  LD      B528  ; L-BendInTurnSw
      AND     B0F21  ; Manual  ModeLampL&Z
      LD      M2324  ; L-Bend  BendTurnAt
      AND     B0F23  ; Auto    ModeLampL&Z
      ORB
      AND     T715  ; L-BendInPush RevTm
      ANI     M2250  ; L-BenderHomeRetnSet
      ANI     Y529  ; L-BendInReturnSv
      OUT     Y528  ; L-BendInTurnSv
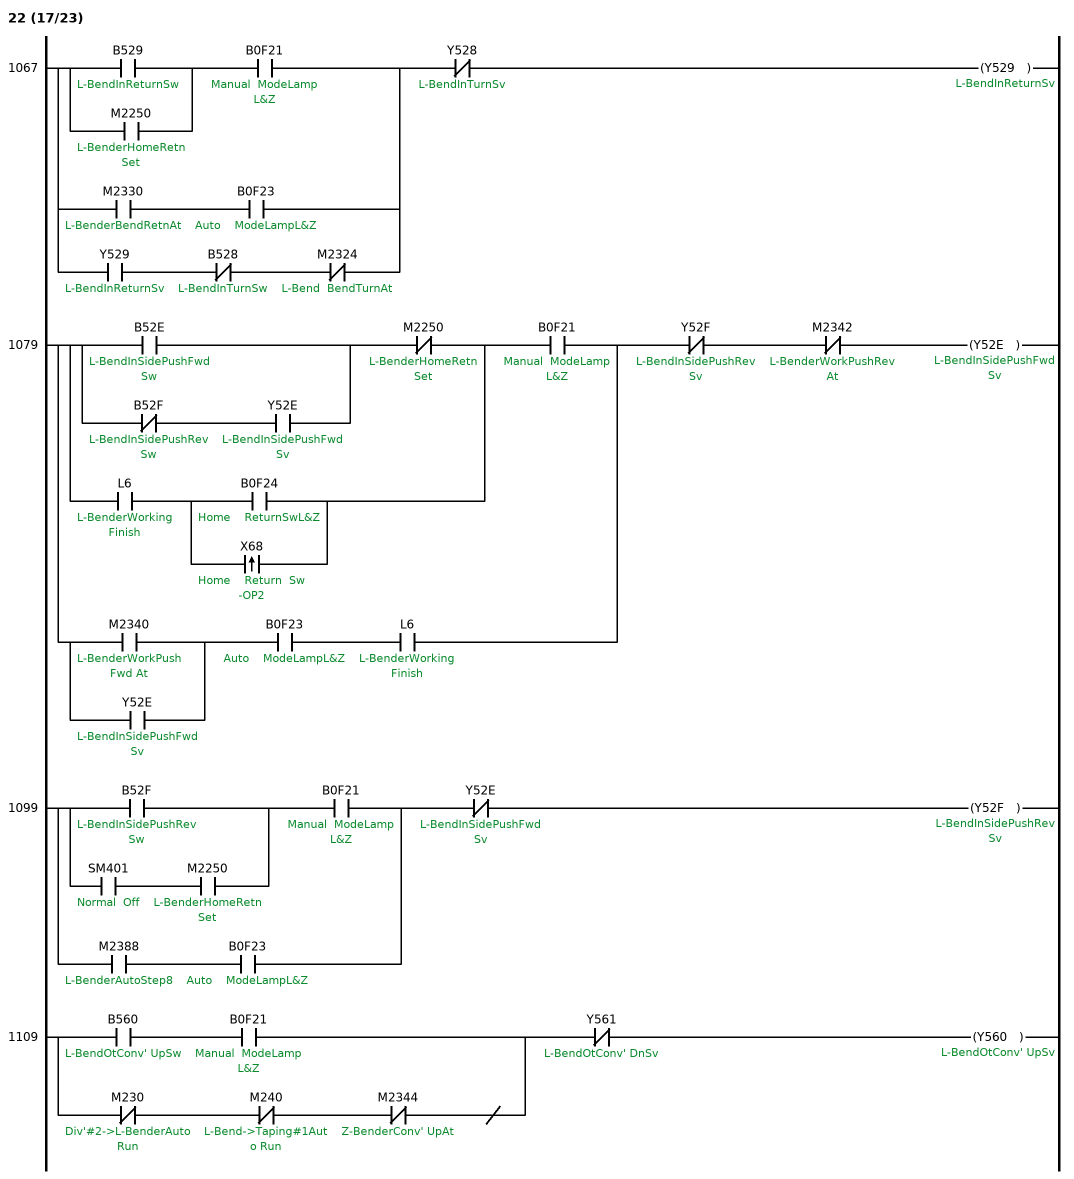
1067  LD      B529  ; L-BendInReturnSw
      OR      M2250  ; L-BenderHomeRetnSet
      AND     B0F21  ; Manual  ModeLampL&Z
      LD      M2330  ; L-BenderBendRetnAt
      AND     B0F23  ; Auto    ModeLampL&Z
      ORB
      LD      Y529  ; L-BendInReturnSv
      ANI     B528  ; L-BendInTurnSw
      ANI     M2324  ; L-Bend  BendTurnAt
      ORB
      ANI     Y528  ; L-BendInTurnSv
      OUT     Y529  ; L-BendInReturnSv
1079  LD      B52E  ; L-BendInSidePushFwd Sw
      LDI     B52F  ; L-BendInSidePushRev Sw
      AND     Y52E  ; L-BendInSidePushFwd Sv
      ORB
      ANI     M2250  ; L-BenderHomeRetnSet
      LD      L6  ; L-BenderWorking Finish
      LD      B0F24  ; Home    ReturnSwL&Z
      ORP     X68  ; Home    Return  Sw -OP2
      ANB
      ORB
      AND     B0F21  ; Manual  ModeLampL&Z
      LD      M2340  ; L-BenderWorkPushFwd At
      OR      Y52E  ; L-BendInSidePushFwd Sv
      AND     B0F23  ; Auto    ModeLampL&Z
      AND     L6  ; L-BenderWorking Finish
      ORB
      ANI     Y52F  ; L-BendInSidePushRevSv
      ANI     M2342  ; L-BenderWorkPushRev At
      OUT     Y52E  ; L-BendInSidePushFwd Sv
1099  LD      B52F  ; L-BendInSidePushRev Sw
      LD      SM401  ; Normal  Off
      AND     M2250  ; L-BenderHomeRetnSet
      ORB
      AND     B0F21  ; Manual  ModeLampL&Z
      LD      M2388  ; L-BenderAutoStep8
      AND     B0F23  ; Auto    ModeLampL&Z
      ORB
      ANI     Y52E  ; L-BendInSidePushFwd Sv
      OUT     Y52F  ; L-BendInSidePushRevSv
1109  LD      B560  ; L-BendOtConv' UpSw
      AND     B0F21  ; Manual  ModeLampL&Z
      LDI     M230  ; Div'#2->L-BenderAuto Run
      ANI     M240  ; L-Bend->Taping#1Auto Run
      ANI     M2344  ; Z-BenderConv' UpAt
      INV
      ORB
      ANI     Y561  ; L-BendOtConv' DnSv
      OUT     Y560  ; L-BendOtConv' UpSv
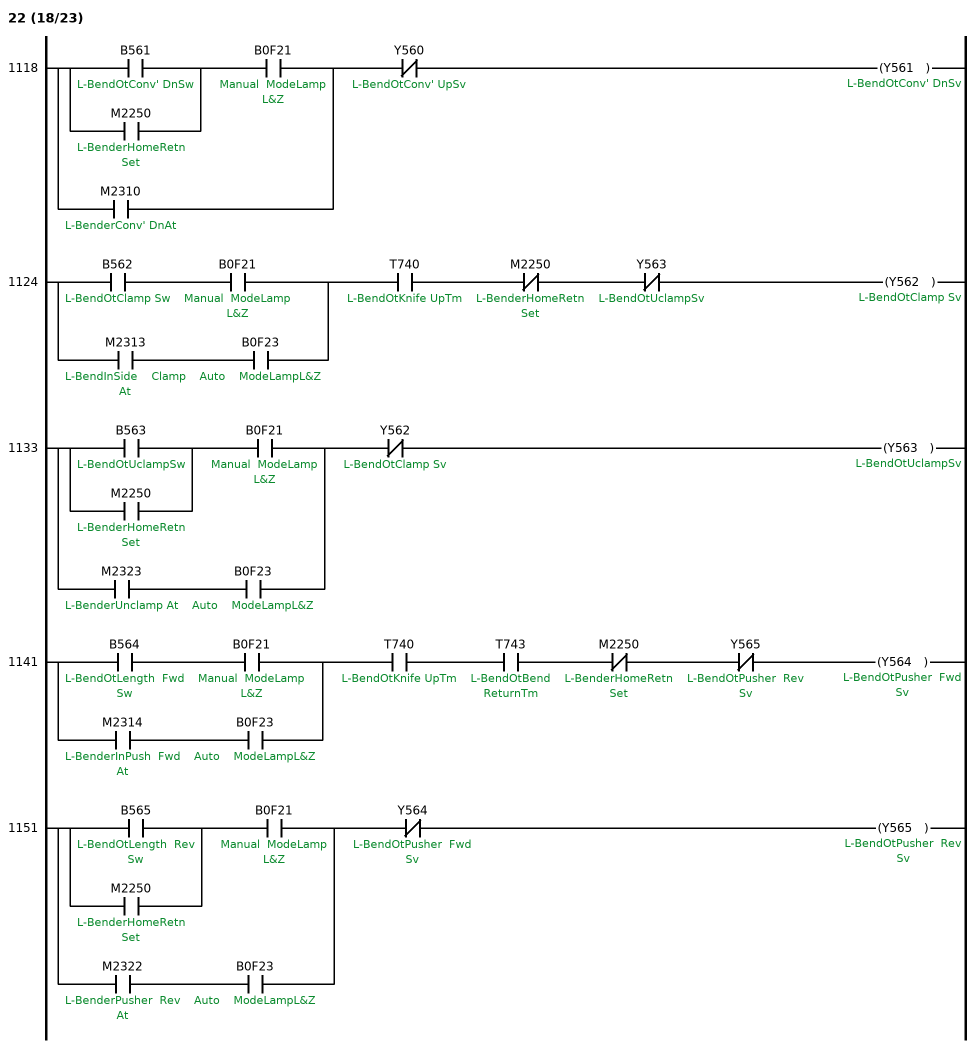
1118  LD      B561  ; L-BendOtConv' DnSw
      OR      M2250  ; L-BenderHomeRetnSet
      AND     B0F21  ; Manual  ModeLampL&Z
      OR      M2310  ; L-BenderConv' DnAt
      ANI     Y560  ; L-BendOtConv' UpSv
      OUT     Y561  ; L-BendOtConv' DnSv
1124  LD      B562  ; L-BendOtClamp Sw
      AND     B0F21  ; Manual  ModeLampL&Z
      LD      M2313  ; L-BendInSide    Clamp At
      AND     B0F23  ; Auto    ModeLampL&Z
      ORB
      AND     T740  ; L-BendOtKnife UpTm
      ANI     M2250  ; L-BenderHomeRetnSet
      ANI     Y563  ; L-BendOtUclampSv
      OUT     Y562  ; L-BendOtClamp Sv
1133  LD      B563  ; L-BendOtUclampSw
      OR      M2250  ; L-BenderHomeRetnSet
      AND     B0F21  ; Manual  ModeLampL&Z
      LD      M2323  ; L-BenderUnclamp At
      AND     B0F23  ; Auto    ModeLampL&Z
      ORB
      ANI     Y562  ; L-BendOtClamp Sv
      OUT     Y563  ; L-BendOtUclampSv
1141  LD      B564  ; L-BendOtLength  Fwd Sw
      AND     B0F21  ; Manual  ModeLampL&Z
      LD      M2314  ; L-BenderInPush  Fwd At
      AND     B0F23  ; Auto    ModeLampL&Z
      ORB
      AND     T740  ; L-BendOtKnife UpTm
      AND     T743  ; L-BendOtBend    ReturnTm
      ANI     M2250  ; L-BenderHomeRetnSet
      ANI     Y565  ; L-BendOtPusher  Rev Sv
      OUT     Y564  ; L-BendOtPusher  Fwd Sv
1151  LD      B565  ; L-BendOtLength  Rev Sw
      OR      M2250  ; L-BenderHomeRetnSet
      AND     B0F21  ; Manual  ModeLampL&Z
      LD      M2322  ; L-BenderPusher  Rev At
      AND     B0F23  ; Auto    ModeLampL&Z
      ORB
      ANI     Y564  ; L-BendOtPusher  Fwd Sv
      OUT     Y565  ; L-BendOtPusher  Rev Sv
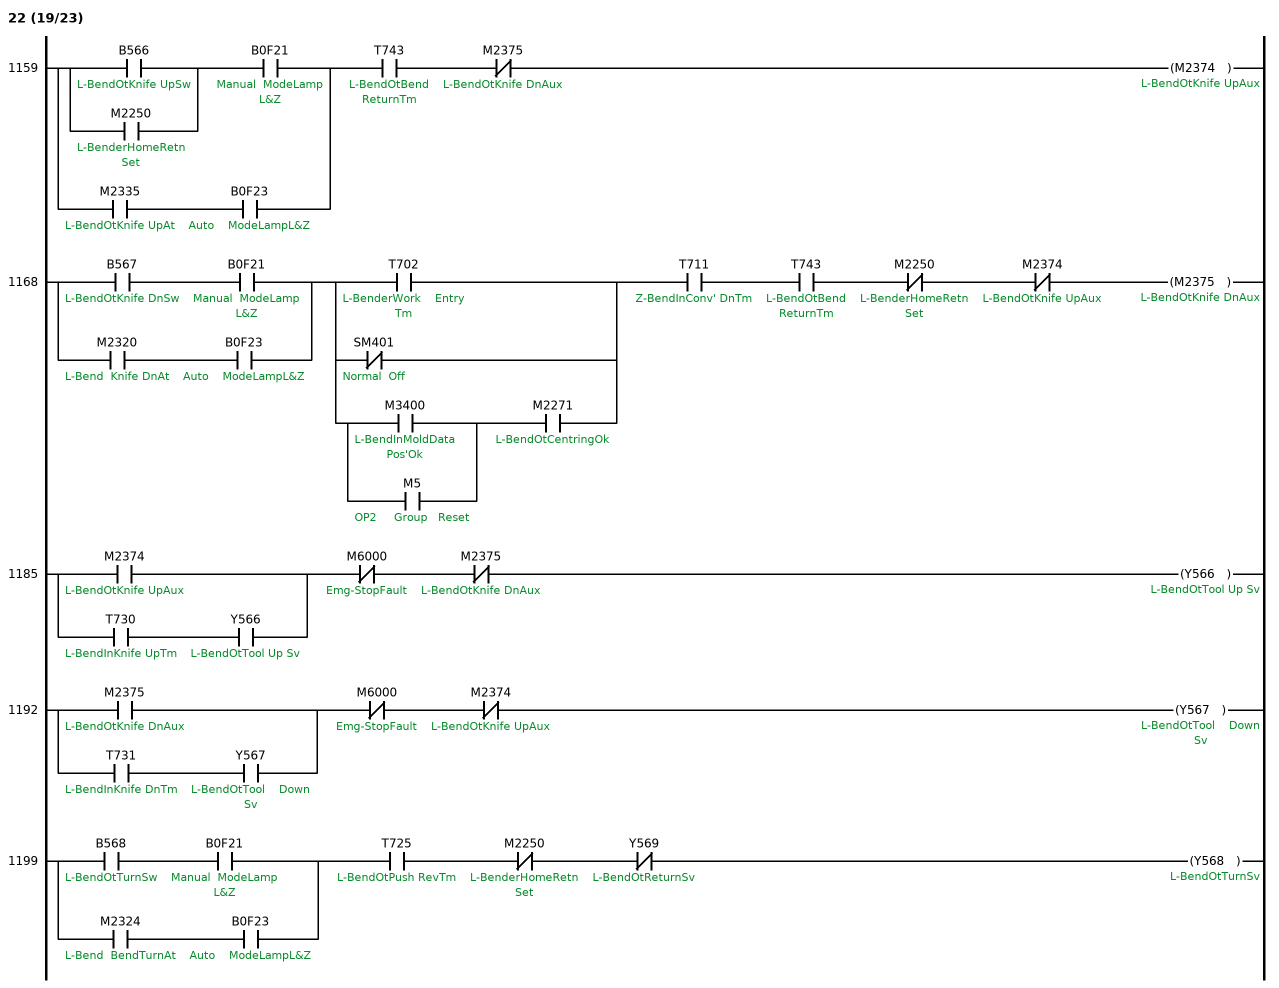
1159  LD      B566  ; L-BendOtKnife UpSw
      OR      M2250  ; L-BenderHomeRetnSet
      AND     B0F21  ; Manual  ModeLampL&Z
      LD      M2335  ; L-BendOtKnife UpAt
      AND     B0F23  ; Auto    ModeLampL&Z
      ORB
      AND     T743  ; L-BendOtBend    ReturnTm
      ANI     M2375  ; L-BendOtKnife DnAux
      OUT     M2374  ; L-BendOtKnife UpAux
1168  LD      B567  ; L-BendOtKnife DnSw
      AND     B0F21  ; Manual  ModeLampL&Z
      LD      M2320  ; L-Bend  Knife DnAt
      AND     B0F23  ; Auto    ModeLampL&Z
      ORB
      LD      T702  ; L-BenderWork    Entry Tm
      ORI     SM401  ; Normal  Off
      LD      M3400  ; L-BendInMoldDataPos'Ok
      OR      M5  ; OP2     Group   Reset
      AND     M2271  ; L-BendOtCentringOk
      ORB
      ANB
      AND     T711  ; Z-BendInConv' DnTm
      AND     T743  ; L-BendOtBend    ReturnTm
      ANI     M2250  ; L-BenderHomeRetnSet
      ANI     M2374  ; L-BendOtKnife UpAux
      OUT     M2375  ; L-BendOtKnife DnAux
1185  LD      M2374  ; L-BendOtKnife UpAux
      LD      T730  ; L-BendInKnife UpTm
      AND     Y566  ; L-BendOtTool Up Sv
      ORB
      ANI     M6000  ; Emg-StopFault
      ANI     M2375  ; L-BendOtKnife DnAux
      OUT     Y566  ; L-BendOtTool Up Sv
1192  LD      M2375  ; L-BendOtKnife DnAux
      LD      T731  ; L-BendInKnife DnTm
      AND     Y567  ; L-BendOtTool    Down Sv
      ORB
      ANI     M6000  ; Emg-StopFault
      ANI     M2374  ; L-BendOtKnife UpAux
      OUT     Y567  ; L-BendOtTool    Down Sv
1199  LD      B568  ; L-BendOtTurnSw
      AND     B0F21  ; Manual  ModeLampL&Z
      LD      M2324  ; L-Bend  BendTurnAt
      AND     B0F23  ; Auto    ModeLampL&Z
      ORB
      AND     T725  ; L-BendOtPush RevTm
      ANI     M2250  ; L-BenderHomeRetnSet
      ANI     Y569  ; L-BendOtReturnSv
      OUT     Y568  ; L-BendOtTurnSv
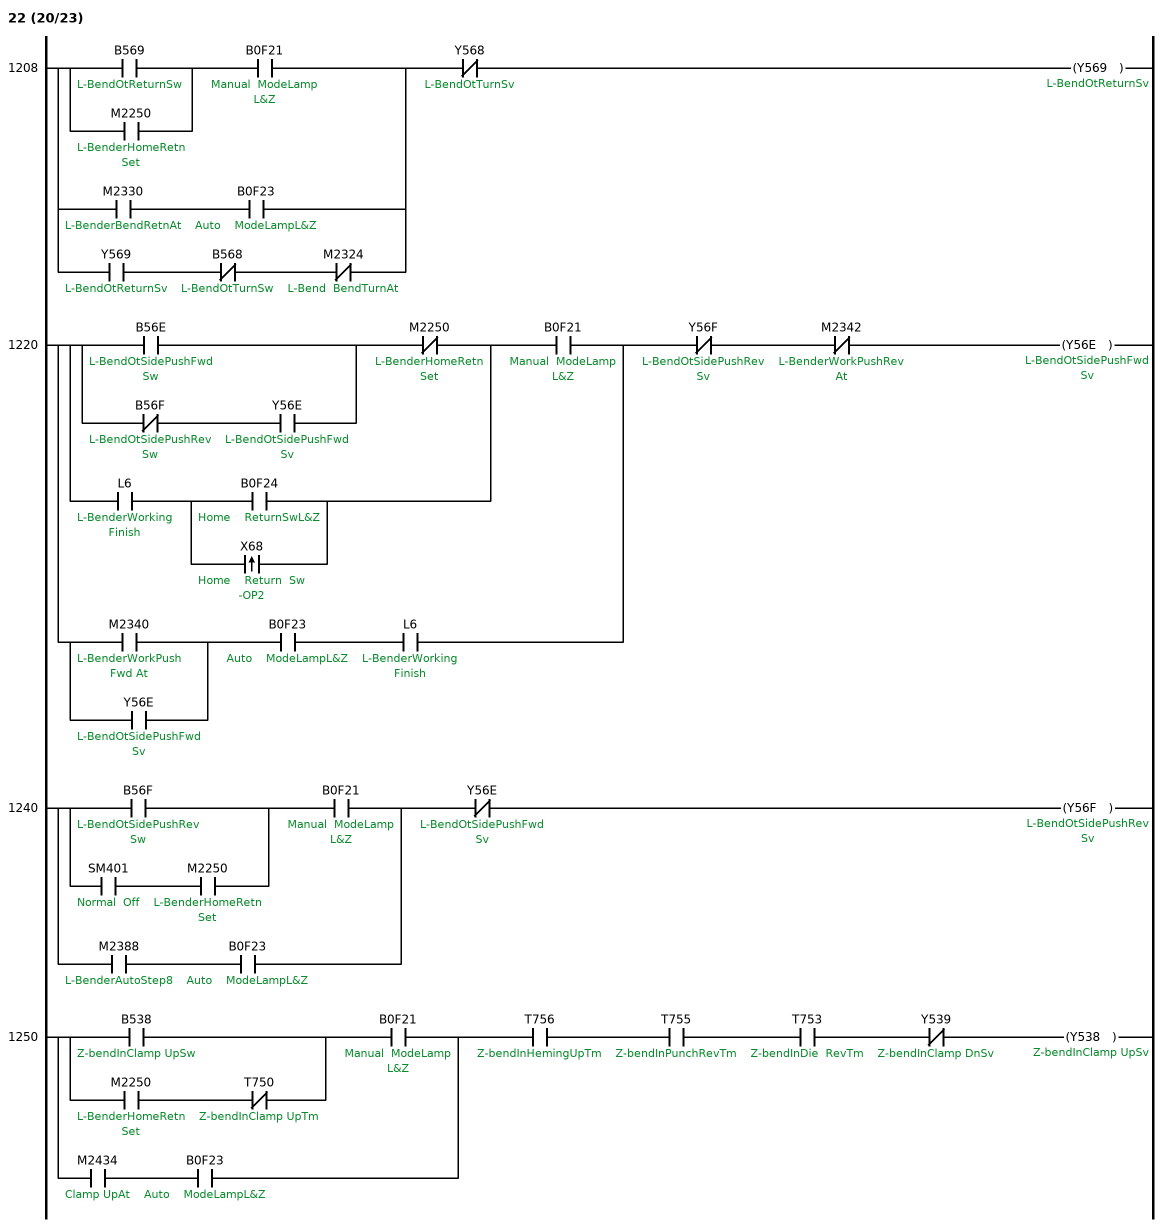
1208  LD      B569  ; L-BendOtReturnSw
      OR      M2250  ; L-BenderHomeRetnSet
      AND     B0F21  ; Manual  ModeLampL&Z
      LD      M2330  ; L-BenderBendRetnAt
      AND     B0F23  ; Auto    ModeLampL&Z
      ORB
      LD      Y569  ; L-BendOtReturnSv
      ANI     B568  ; L-BendOtTurnSw
      ANI     M2324  ; L-Bend  BendTurnAt
      ORB
      ANI     Y568  ; L-BendOtTurnSv
      OUT     Y569  ; L-BendOtReturnSv
1220  LD      B56E  ; L-BendOtSidePushFwd Sw
      LDI     B56F  ; L-BendOtSidePushRev Sw
      AND     Y56E  ; L-BendOtSidePushFwd Sv
      ORB
      ANI     M2250  ; L-BenderHomeRetnSet
      LD      L6  ; L-BenderWorking Finish
      LD      B0F24  ; Home    ReturnSwL&Z
      ORP     X68  ; Home    Return  Sw -OP2
      ANB
      ORB
      AND     B0F21  ; Manual  ModeLampL&Z
      LD      M2340  ; L-BenderWorkPushFwd At
      OR      Y56E  ; L-BendOtSidePushFwd Sv
      AND     B0F23  ; Auto    ModeLampL&Z
      AND     L6  ; L-BenderWorking Finish
      ORB
      ANI     Y56F  ; L-BendOtSidePushRev Sv
      ANI     M2342  ; L-BenderWorkPushRev At
      OUT     Y56E  ; L-BendOtSidePushFwd Sv
1240  LD      B56F  ; L-BendOtSidePushRev Sw
      LD      SM401  ; Normal  Off
      AND     M2250  ; L-BenderHomeRetnSet
      ORB
      AND     B0F21  ; Manual  ModeLampL&Z
      LD      M2388  ; L-BenderAutoStep8
      AND     B0F23  ; Auto    ModeLampL&Z
      ORB
      ANI     Y56E  ; L-BendOtSidePushFwd Sv
      OUT     Y56F  ; L-BendOtSidePushRev Sv
1250  LD      B538  ; Z-bendInClamp UpSw
      LD      M2250  ; L-BenderHomeRetnSet
      ANI     T750  ; Z-bendInClamp UpTm
      ORB
      AND     B0F21  ; Manual  ModeLampL&Z
      LD      M2434  ; Clamp UpAt
      AND     B0F23  ; Auto    ModeLampL&Z
      ORB
      AND     T756  ; Z-bendInHemingUpTm
      AND     T755  ; Z-bendInPunchRevTm
      AND     T753  ; Z-bendInDie  RevTm
      ANI     Y539  ; Z-bendInClamp DnSv
      OUT     Y538  ; Z-bendInClamp UpSv
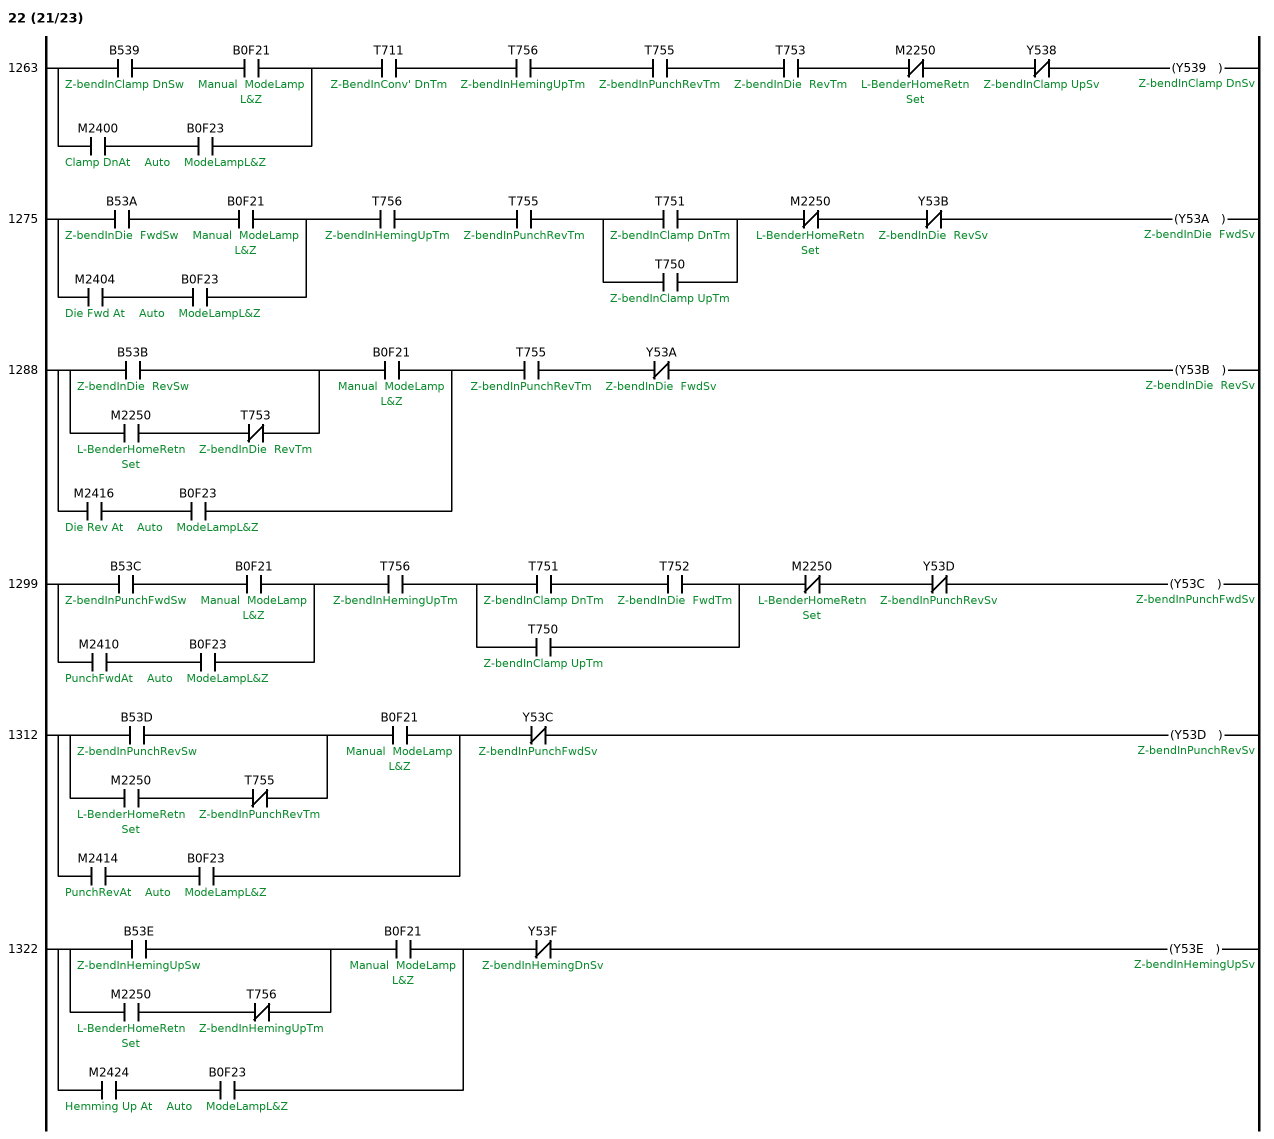
1263  LD      B539  ; Z-bendInClamp DnSw
      AND     B0F21  ; Manual  ModeLampL&Z
      LD      M2400  ; Clamp DnAt
      AND     B0F23  ; Auto    ModeLampL&Z
      ORB
      AND     T711  ; Z-BendInConv' DnTm
      AND     T756  ; Z-bendInHemingUpTm
      AND     T755  ; Z-bendInPunchRevTm
      AND     T753  ; Z-bendInDie  RevTm
      ANI     M2250  ; L-BenderHomeRetnSet
      ANI     Y538  ; Z-bendInClamp UpSv
      OUT     Y539  ; Z-bendInClamp DnSv
1275  LD      B53A  ; Z-bendInDie  FwdSw
      AND     B0F21  ; Manual  ModeLampL&Z
      LD      M2404  ; Die Fwd At
      AND     B0F23  ; Auto    ModeLampL&Z
      ORB
      AND     T756  ; Z-bendInHemingUpTm
      AND     T755  ; Z-bendInPunchRevTm
      LD      T751  ; Z-bendInClamp DnTm
      OR      T750  ; Z-bendInClamp UpTm
      ANB
      ANI     M2250  ; L-BenderHomeRetnSet
      ANI     Y53B  ; Z-bendInDie  RevSv
      OUT     Y53A  ; Z-bendInDie  FwdSv
1288  LD      B53B  ; Z-bendInDie  RevSw
      LD      M2250  ; L-BenderHomeRetnSet
      ANI     T753  ; Z-bendInDie  RevTm
      ORB
      AND     B0F21  ; Manual  ModeLampL&Z
      LD      M2416  ; Die Rev At
      AND     B0F23  ; Auto    ModeLampL&Z
      ORB
      AND     T755  ; Z-bendInPunchRevTm
      ANI     Y53A  ; Z-bendInDie  FwdSv
      OUT     Y53B  ; Z-bendInDie  RevSv
1299  LD      B53C  ; Z-bendInPunchFwdSw
      AND     B0F21  ; Manual  ModeLampL&Z
      LD      M2410  ; PunchFwdAt
      AND     B0F23  ; Auto    ModeLampL&Z
      ORB
      AND     T756  ; Z-bendInHemingUpTm
      LD      T751  ; Z-bendInClamp DnTm
      AND     T752  ; Z-bendInDie  FwdTm
      OR      T750  ; Z-bendInClamp UpTm
      ANB
      ANI     M2250  ; L-BenderHomeRetnSet
      ANI     Y53D  ; Z-bendInPunchRevSv
      OUT     Y53C  ; Z-bendInPunchFwdSv
1312  LD      B53D  ; Z-bendInPunchRevSw
      LD      M2250  ; L-BenderHomeRetnSet
      ANI     T755  ; Z-bendInPunchRevTm
      ORB
      AND     B0F21  ; Manual  ModeLampL&Z
      LD      M2414  ; PunchRevAt
      AND     B0F23  ; Auto    ModeLampL&Z
      ORB
      ANI     Y53C  ; Z-bendInPunchFwdSv
      OUT     Y53D  ; Z-bendInPunchRevSv
1322  LD      B53E  ; Z-bendInHemingUpSw
      LD      M2250  ; L-BenderHomeRetnSet
      ANI     T756  ; Z-bendInHemingUpTm
      ORB
      AND     B0F21  ; Manual  ModeLampL&Z
      LD      M2424  ; Hemming Up At
      AND     B0F23  ; Auto    ModeLampL&Z
      ORB
      ANI     Y53F  ; Z-bendInHemingDnSv
      OUT     Y53E  ; Z-bendInHemingUpSv
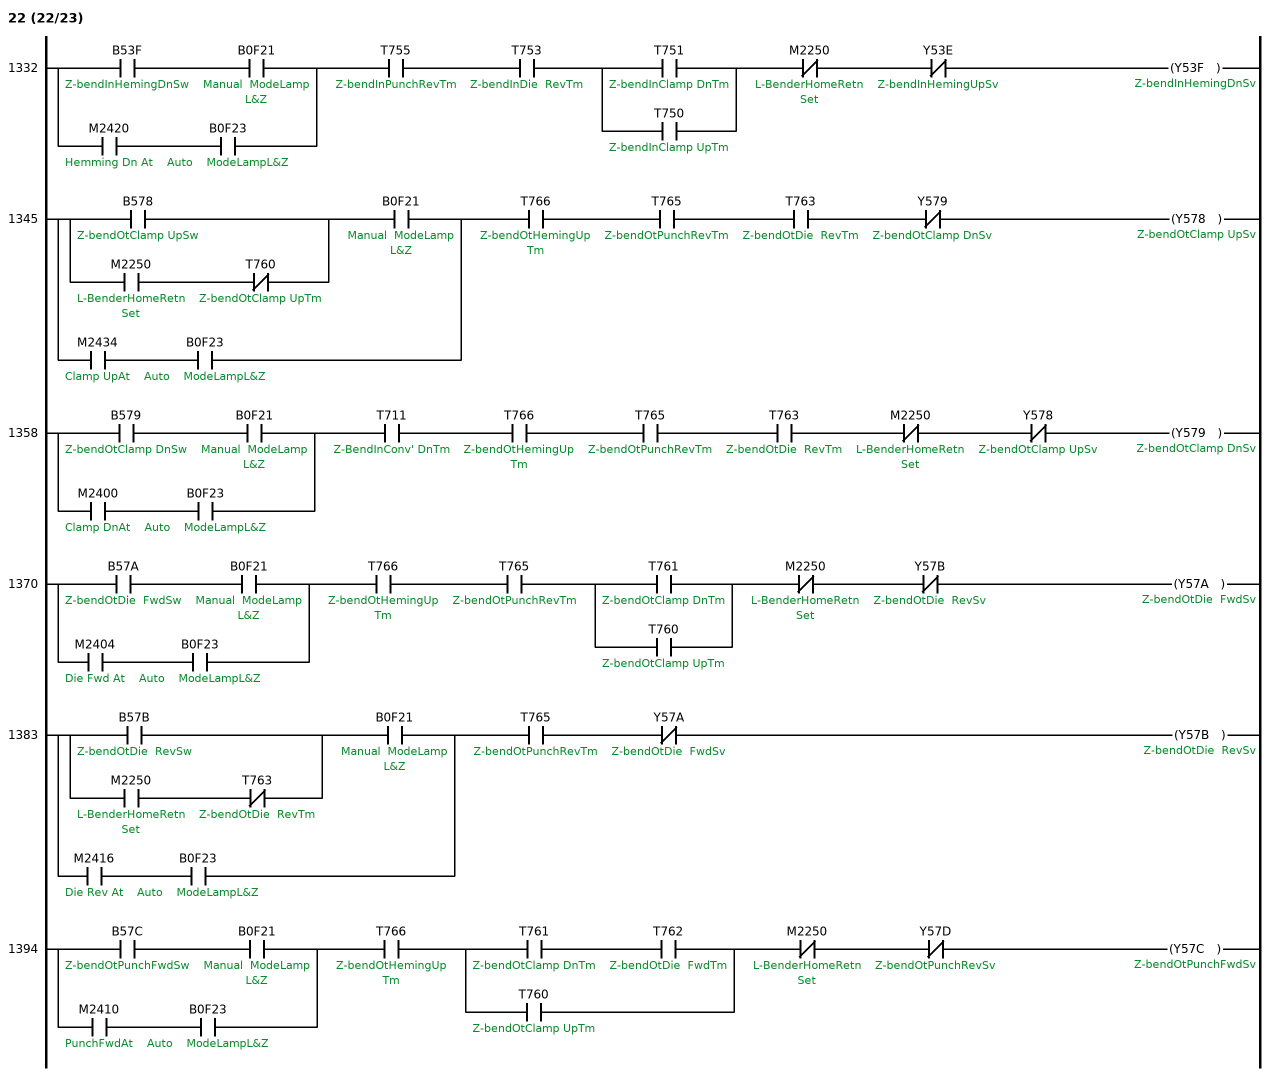
1332  LD      B53F  ; Z-bendInHemingDnSw
      AND     B0F21  ; Manual  ModeLampL&Z
      LD      M2420  ; Hemming Dn At
      AND     B0F23  ; Auto    ModeLampL&Z
      ORB
      AND     T755  ; Z-bendInPunchRevTm
      AND     T753  ; Z-bendInDie  RevTm
      LD      T751  ; Z-bendInClamp DnTm
      OR      T750  ; Z-bendInClamp UpTm
      ANB
      ANI     M2250  ; L-BenderHomeRetnSet
      ANI     Y53E  ; Z-bendInHemingUpSv
      OUT     Y53F  ; Z-bendInHemingDnSv
1345  LD      B578  ; Z-bendOtClamp UpSw
      LD      M2250  ; L-BenderHomeRetnSet
      ANI     T760  ; Z-bendOtClamp UpTm
      ORB
      AND     B0F21  ; Manual  ModeLampL&Z
      LD      M2434  ; Clamp UpAt
      AND     B0F23  ; Auto    ModeLampL&Z
      ORB
      AND     T766  ; Z-bendOtHemingUpTm
      AND     T765  ; Z-bendOtPunchRevTm
      AND     T763  ; Z-bendOtDie  RevTm
      ANI     Y579  ; Z-bendOtClamp DnSv
      OUT     Y578  ; Z-bendOtClamp UpSv
1358  LD      B579  ; Z-bendOtClamp DnSw
      AND     B0F21  ; Manual  ModeLampL&Z
      LD      M2400  ; Clamp DnAt
      AND     B0F23  ; Auto    ModeLampL&Z
      ORB
      AND     T711  ; Z-BendInConv' DnTm
      AND     T766  ; Z-bendOtHemingUpTm
      AND     T765  ; Z-bendOtPunchRevTm
      AND     T763  ; Z-bendOtDie  RevTm
      ANI     M2250  ; L-BenderHomeRetnSet
      ANI     Y578  ; Z-bendOtClamp UpSv
      OUT     Y579  ; Z-bendOtClamp DnSv
1370  LD      B57A  ; Z-bendOtDie  FwdSw
      AND     B0F21  ; Manual  ModeLampL&Z
      LD      M2404  ; Die Fwd At
      AND     B0F23  ; Auto    ModeLampL&Z
      ORB
      AND     T766  ; Z-bendOtHemingUpTm
      AND     T765  ; Z-bendOtPunchRevTm
      LD      T761  ; Z-bendOtClamp DnTm
      OR      T760  ; Z-bendOtClamp UpTm
      ANB
      ANI     M2250  ; L-BenderHomeRetnSet
      ANI     Y57B  ; Z-bendOtDie  RevSv
      OUT     Y57A  ; Z-bendOtDie  FwdSv
1383  LD      B57B  ; Z-bendOtDie  RevSw
      LD      M2250  ; L-BenderHomeRetnSet
      ANI     T763  ; Z-bendOtDie  RevTm
      ORB
      AND     B0F21  ; Manual  ModeLampL&Z
      LD      M2416  ; Die Rev At
      AND     B0F23  ; Auto    ModeLampL&Z
      ORB
      AND     T765  ; Z-bendOtPunchRevTm
      ANI     Y57A  ; Z-bendOtDie  FwdSv
      OUT     Y57B  ; Z-bendOtDie  RevSv
1394  LD      B57C  ; Z-bendOtPunchFwdSw
      AND     B0F21  ; Manual  ModeLampL&Z
      LD      M2410  ; PunchFwdAt
      AND     B0F23  ; Auto    ModeLampL&Z
      ORB
      AND     T766  ; Z-bendOtHemingUpTm
      LD      T761  ; Z-bendOtClamp DnTm
      AND     T762  ; Z-bendOtDie  FwdTm
      OR      T760  ; Z-bendOtClamp UpTm
      ANB
      ANI     M2250  ; L-BenderHomeRetnSet
      ANI     Y57D  ; Z-bendOtPunchRevSv
      OUT     Y57C  ; Z-bendOtPunchFwdSv
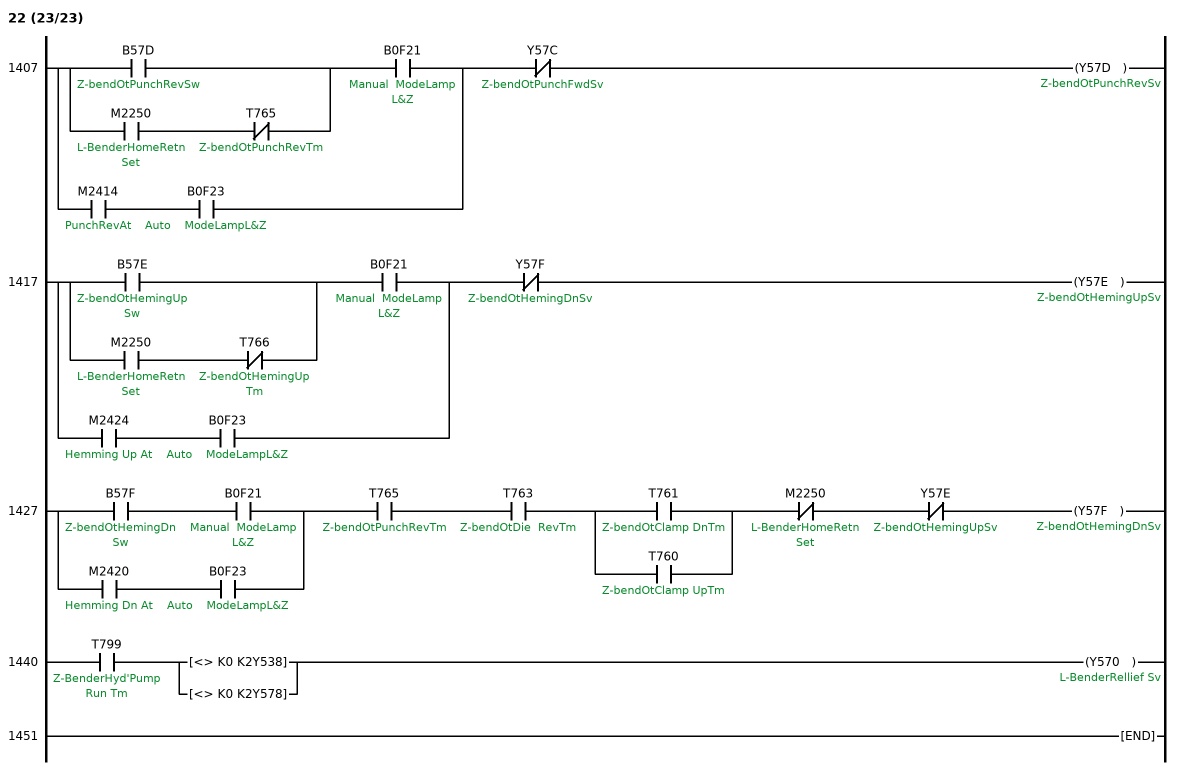
1407  LD      B57D  ; Z-bendOtPunchRevSw
      LD      M2250  ; L-BenderHomeRetnSet
      ANI     T765  ; Z-bendOtPunchRevTm
      ORB
      AND     B0F21  ; Manual  ModeLampL&Z
      LD      M2414  ; PunchRevAt
      AND     B0F23  ; Auto    ModeLampL&Z
      ORB
      ANI     Y57C  ; Z-bendOtPunchFwdSv
      OUT     Y57D  ; Z-bendOtPunchRevSv
1417  LD      B57E  ; Z-bendOtHemingUpSw
      LD      M2250  ; L-BenderHomeRetnSet
      ANI     T766  ; Z-bendOtHemingUpTm
      ORB
      AND     B0F21  ; Manual  ModeLampL&Z
      LD      M2424  ; Hemming Up At
      AND     B0F23  ; Auto    ModeLampL&Z
      ORB
      ANI     Y57F  ; Z-bendOtHemingDnSv
      OUT     Y57E  ; Z-bendOtHemingUpSv
1427  LD      B57F  ; Z-bendOtHemingDnSw
      AND     B0F21  ; Manual  ModeLampL&Z
      LD      M2420  ; Hemming Dn At
      AND     B0F23  ; Auto    ModeLampL&Z
      ORB
      AND     T765  ; Z-bendOtPunchRevTm
      AND     T763  ; Z-bendOtDie  RevTm
      LD      T761  ; Z-bendOtClamp DnTm
      OR      T760  ; Z-bendOtClamp UpTm
      ANB
      ANI     M2250  ; L-BenderHomeRetnSet
      ANI     Y57E  ; Z-bendOtHemingUpSv
      OUT     Y57F  ; Z-bendOtHemingDnSv
1440  LD      T799  ; Z-BenderHyd'PumpRun Tm
      LD<>    K0 K2Y538  ; Z-bendInClamp UpSv
      OR<>    K0 K2Y578  ; Z-bendOtClamp UpSv
      ANB
      OUT     Y570  ; L-BenderRellief Sv
1451  END
END_PROGRAM

PROGRAM 23  // Taping Conveyor
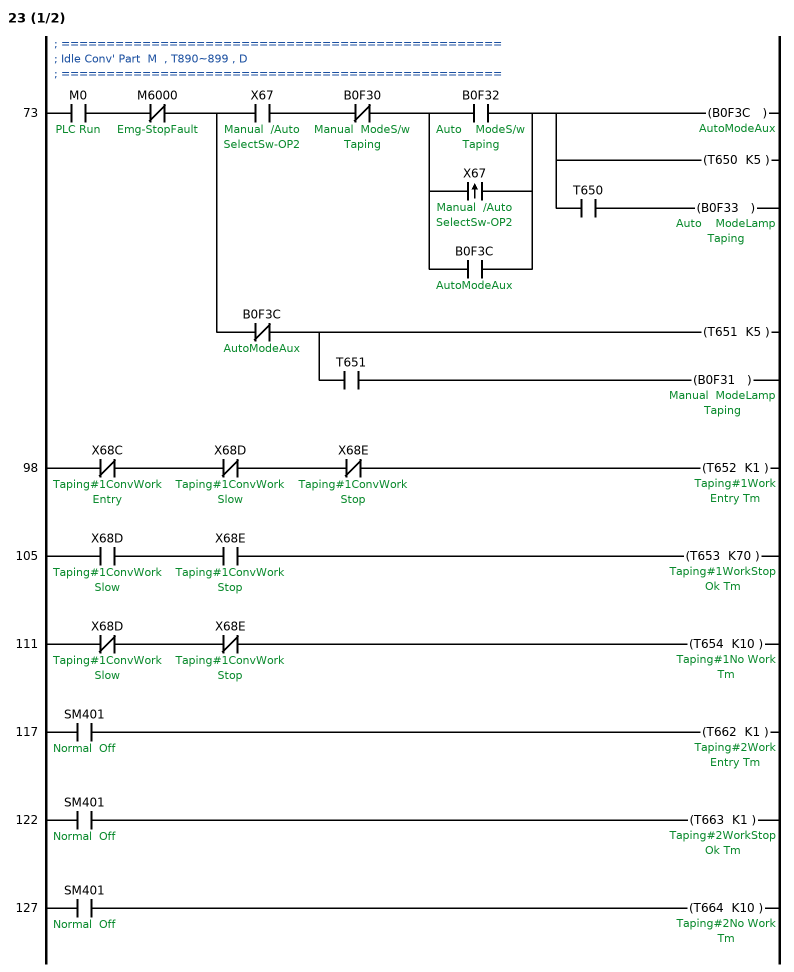
; =================================================
; Idle Conv' Part  M  , T890~899 , D
; =================================================
73    LD      M0  ; PLC Run
      ANI     M6000  ; Emg-StopFault
      MPS
      AND     X67  ; Manual  /Auto   SelectSw-OP2
      ANI     B0F30  ; Manual  ModeS/w Taping
      LD      B0F32  ; Auto    ModeS/w Taping
      ORP     X67  ; Manual  /Auto   SelectSw-OP2
      OR      B0F3C  ; AutoModeAux
      ANB
      OUT     B0F3C  ; AutoModeAux
      OUT     T650 K5
      AND     T650
      OUT     B0F33  ; Auto    ModeLampTaping
      MPP
      ANI     B0F3C  ; AutoModeAux
      OUT     T651 K5
      AND     T651
      OUT     B0F31  ; Manual  ModeLampTaping
98    LDI     X68C  ; Taping#1ConvWorkEntry
      ANI     X68D  ; Taping#1ConvWorkSlow
      ANI     X68E  ; Taping#1ConvWorkStop
      OUT     T652 K1  ; Taping#1Work    Entry Tm
105   LD      X68D  ; Taping#1ConvWorkSlow
      AND     X68E  ; Taping#1ConvWorkStop
      OUT     T653 K70  ; Taping#1WorkStopOk Tm
111   LDI     X68D  ; Taping#1ConvWorkSlow
      ANI     X68E  ; Taping#1ConvWorkStop
      OUT     T654 K10  ; Taping#1No Work Tm
117   LD      SM401  ; Normal  Off
      OUT     T662 K1  ; Taping#2Work    Entry Tm
122   LD      SM401  ; Normal  Off
      OUT     T663 K1  ; Taping#2WorkStopOk Tm
127   LD      SM401  ; Normal  Off
      OUT     T664 K10  ; Taping#2No Work Tm
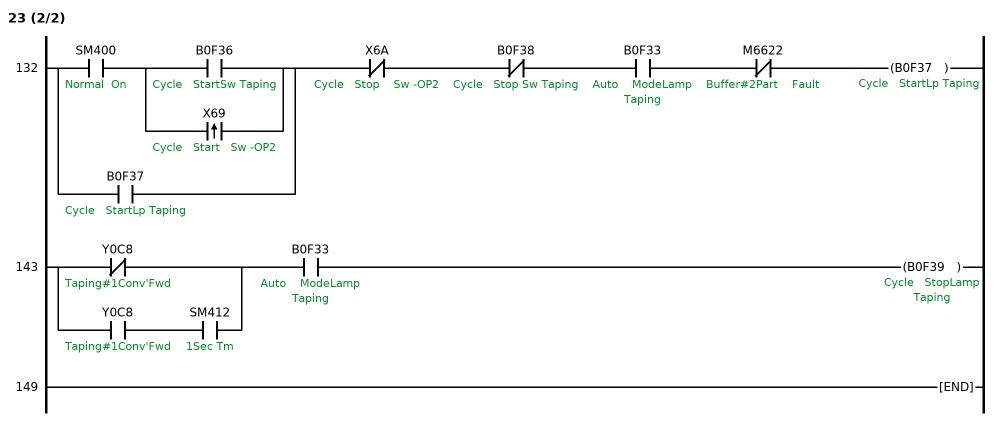
132   LD      SM400  ; Normal  On
      LD      B0F36  ; Cycle   StartSw Taping
      ORP     X69  ; Cycle   Start   Sw -OP2
      ANB
      OR      B0F37  ; Cycle   StartLp Taping
      ANI     X6A  ; Cycle   Stop    Sw -OP2
      ANI     B0F38  ; Cycle   Stop Sw Taping
      AND     B0F33  ; Auto    ModeLampTaping
      ANI     M6622  ; Buffer#2Part    Fault
      OUT     B0F37  ; Cycle   StartLp Taping
143   LDI     Y0C8  ; Taping#1Conv'Fwd
      LD      Y0C8  ; Taping#1Conv'Fwd
      AND     SM412  ; 1Sec Tm
      ORB
      AND     B0F33  ; Auto    ModeLampTaping
      OUT     B0F39  ; Cycle   StopLampTaping
149   END
END_PROGRAM

PROGRAM 24  // U-Bender
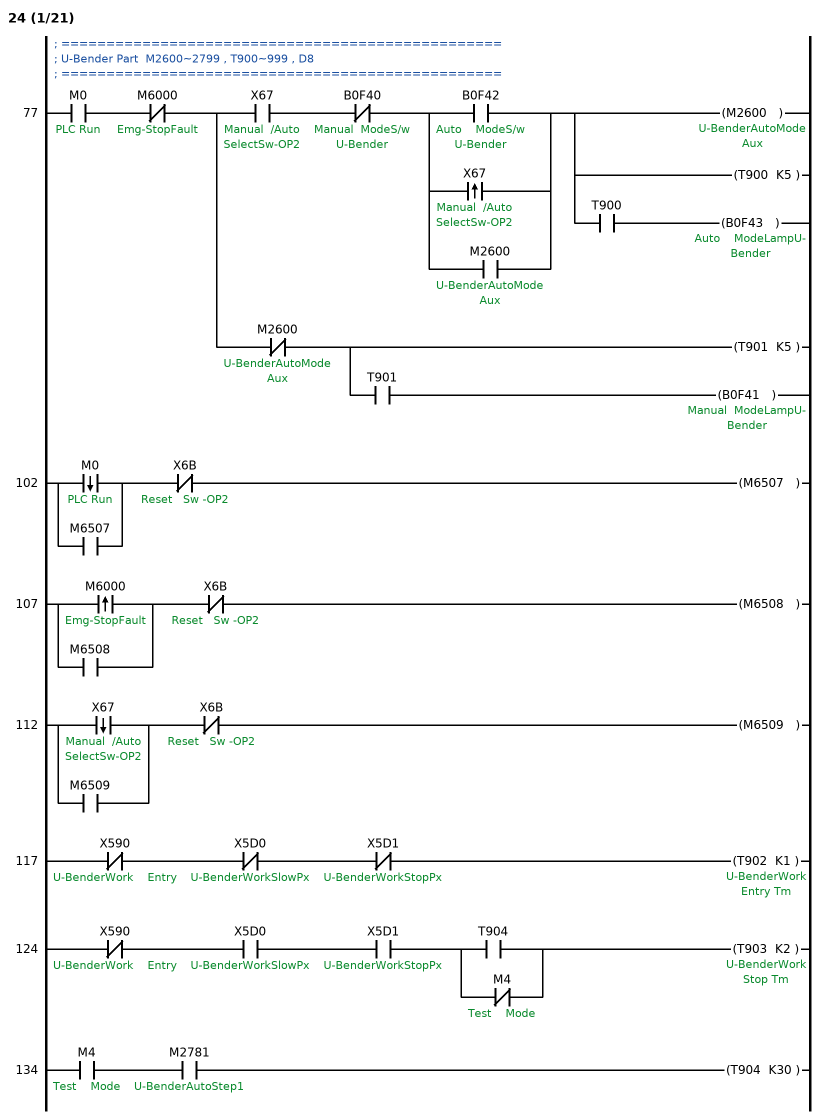
; =================================================
; U-Bender Part  M2600~2799 , T900~999 , D8
; =================================================
77    LD      M0  ; PLC Run
      ANI     M6000  ; Emg-StopFault
      MPS
      AND     X67  ; Manual  /Auto   SelectSw-OP2
      ANI     B0F40  ; Manual  ModeS/w U-Bender
      LD      B0F42  ; Auto    ModeS/w U-Bender
      ORP     X67  ; Manual  /Auto   SelectSw-OP2
      OR      M2600  ; U-BenderAutoModeAux
      ANB
      OUT     M2600  ; U-BenderAutoModeAux
      OUT     T900 K5
      AND     T900
      OUT     B0F43  ; Auto    ModeLampU-Bender
      MPP
      ANI     M2600  ; U-BenderAutoModeAux
      OUT     T901 K5
      AND     T901
      OUT     B0F41  ; Manual  ModeLampU-Bender
102   LDF     M0  ; PLC Run
      OR      M6507
      ANI     X6B  ; Reset   Sw -OP2
      OUT     M6507
107   LDP     M6000  ; Emg-StopFault
      OR      M6508
      ANI     X6B  ; Reset   Sw -OP2
      OUT     M6508
112   LDF     X67  ; Manual  /Auto   SelectSw-OP2
      OR      M6509
      ANI     X6B  ; Reset   Sw -OP2
      OUT     M6509
117   LDI     X590  ; U-BenderWork    Entry
      ANI     X5D0  ; U-BenderWorkSlowPx
      ANI     X5D1  ; U-BenderWorkStopPx
      OUT     T902 K1  ; U-BenderWork    Entry Tm
124   LDI     X590  ; U-BenderWork    Entry
      AND     X5D0  ; U-BenderWorkSlowPx
      AND     X5D1  ; U-BenderWorkStopPx
      LD      T904
      ORI     M4  ; Test    Mode
      ANB
      OUT     T903 K2  ; U-BenderWork    Stop Tm
134   LD      M4  ; Test    Mode
      AND     M2781  ; U-BenderAutoStep1
      OUT     T904 K30
